# B&R Automation Studio project vibratorControlWithCurrentController (part 11)

#### producing.st
```iecst
ACTION producing:

	CASE em.state OF

		STATE_STARTING:

			em.cmd.sc := em.status.parent.state = STATE_STOPPING;

			CASE em.substate OF
				0:
					em.description := '';

					IF (NOT this.newRecipeLoaded AND interface.status.teachingDone AND this.brickCountTeached = recipe.brickCount) OR interface.cmd.skipTeach OR this.hmi.capconModeOff THEN
						interface.status.teachingDone := TRUE;
						brdkStrMemSet(ADR(this.pctFromMeanToLimit),0,SIZEOF(this.pctFromMeanToLimit));
						bufferIdxCounter :=0;
						this.MTDataStatistics_Teach(Enable:=FALSE);
						this.MTFilterMovingAverage_0(Enable:=FALSE);
						this.TeachIntegral_0.Enable := FALSE;
						this.TeachIntegral_0();
						em.substate := 100;
					ELSE
						interface.status.wingStartBrickNOK	:= TRUE;
						interface.parameter.teachBrickCount := 0;
						gCapconInterface.status.teachingDone := FALSE;
						gUpperFlapInterface.cmd.resetStatistics := TRUE; //
						gBottomFlapInterface.cmd.resetCassetteWaitTime := TRUE;
						brdkStrMemSet(ADR(this.pctFromMeanToLimit),0,SIZEOF(this.pctFromMeanToLimit));
						bufferIdxCounter :=0;
						this.countGoodPortionForTeach := 0;
						this.MTDataStatistics_1(Enable:=FALSE);
						this.MTDataStatistics_0(Enable:=FALSE);
						this.MTDataStatistics_Teach(Enable:=FALSE);
						this.MTFilterMovingAverage_0(Enable:=FALSE);
						this.TeachIntegral_0.Enable := FALSE;
						this.TeachIntegral_0();
						this.noAdaptiveTeaching := 0;
						interface.status.cycleTimeAutoMode := 0;
						gBeltInterface.cmd.cycleTimeCount := 0;
						this.MTFilterMovingAverage_1.Enable := FALSE;
						this.MTFilterMovingAverage_1();
						//always delete statistics before a new teach.
						resetStatistics;
						em.substate := 10;
					END_IF

				10:
					em.description := 'wait for wing to be ready';

					IF interface.cmd.wingReady OR interface.cmd.wingRequest THEN
						interface.status.ready := TRUE;
						em.substate := 20;
					END_IF

				20:
					em.description := 'wait for belt to feed bricks';

					IF gBeltInterface.status.dropBrickDone THEN
						interface.status.ready := FALSE;
						em.substate := 30;
					END_IF

				30:
					em.description := 'wait to see if brick is falling';

					this.TON_waitTime.IN := TRUE;
					this.TON_waitTime.PT := T#400ms;
					this.TON_waitTime();

					interface.status.wingStart := this.TON_waitTime.ET >= T#300ms;

					IF this.TON_waitTime.Q AND NOT interface.status.brickDetected THEN
						this.TON_waitTime.IN := FALSE;
						this.TON_waitTime();
						interface.status.wingStartBrickNOK := TRUE;
						em.substate := 40;
					END_IF

				40:
					em.description := 'wait for wing ready';

					IF interface.cmd.wingCmdAck OR gMainInterface.status.emptying THEN
						interface.status.wingStart := FALSE;
						interface.status.wingStartBrickNOK := FALSE;
						interface.status.wingStartBrickOK := FALSE;

						this.TeachIntegral_0.Enable 			:= TRUE;
						this.TeachIntegral_0.In 				:= interface.status.integralSum / USINT_TO_REAL(recipe.brickCount);
						this.TeachIntegral_0.BrickCount 		:= recipe.brickCount;
						this.TeachIntegral_0.CapconModeOn 		:= this.hmi.capconModeOn;
						this.TeachIntegral_0.NoPeaks 			:= interface.status.noVerifiedPeaks;
						this.TeachIntegral_0.NoPortions			:= config.portionsAllowTeach;
						this.TeachIntegral_0();

						interface.status.teachIntegral := this.TeachIntegral_0.Out;

						IF this.TeachIntegral_0.Done THEN
							this.TeachIntegral_0.Enable := FALSE;
							this.TeachIntegral_0();
							interface.status.teachingDone := TRUE;
							this.newRecipeLoaded := FALSE;
							em.substate := 100;
						ELSIF this.TeachIntegral_0.Error THEN
							this.TeachIntegral_0.Enable := FALSE;
							this.TeachIntegral_0();
							em.substate := 200;
						ELSE
							em.substate := 10;
						END_IF
					END_IF

				100:
					em.description := 'Wait for bypassCassette OFF';

					IF NOT gMainInterface.line.bypassCassette OR gMainInterface.status.emptying THEN
						em.substate := 110;
					END_IF

				110:
					em.description := 'teaching done';
					this.brickCountTeached := recipe.brickCount;
					em.cmd.sc := TRUE;

				200:
					em.description := 'teaching error';
					this.alarm.teachingError.active := TRUE;
					em.cmd.sc := TRUE;

			END_CASE

			// redo teaching if an empty is started while the reteach is running.
			IF interface.cmd.emptyWhileTeaching THEN
				this.hmi.redoTeaching := TRUE;
				em.cmd.sc := TRUE;
			END_IF

		STATE_EXECUTE:

			this.timeBetweenBricks := this.timeBetweenBricks + em.status.cycleTime;

			CASE em.substate OF
				0:
					em.description := 'wait for wing ready';

					interface.status.waiting := NOT interface.cmd.wingRequest;

					IF interface.cmd.wingRequest AND recipe.brickCount > 0 THEN
						IF recipe.brickCount <> this.brickCountTeached THEN
							this.newRecipeLoaded := TRUE;
						END_IF
						interface.status.ready := TRUE;
						em.cmd.sc := FALSE;
						this.startTime := 0;
						em.substate := 10;
					ELSE
						em.cmd.sc := TRUE;
					END_IF

				10:
					em.description := 'wait for belt to feed bricks';

					IF interface.cmd.wingReady AND this.startTime = 0 THEN
						this.startTime := TIME_TO_UDINT(clock_ms());
					END_IF

					IF gBeltInterface.status.dropBrickDone THEN
						interface.status.ready := FALSE;
						this.brickPresent := FALSE;
						IF this.startTime = 0 THEN
							this.startTime := TIME_TO_UDINT(clock_ms());
						END_IF
						em.substate := 20;
					END_IF

				20:
					em.description := 'wait to see if brick is falling';

					this.TON_waitTime.IN := TRUE;
					this.TON_waitTime.PT := T#400ms; // falltime through capcon is 400ms
					this.TON_waitTime();

					interface.status.wingStart := this.TON_waitTime.ET >= T#250ms;

					IF this.TON_waitTime.Q AND NOT interface.status.brickDetected THEN
						this.TON_waitTime.IN := FALSE;
						this.TON_waitTime();
						interface.status.wingStart := TRUE;

						em.substate := 30;
					END_IF

				30:
					em.description := 'validate brick';

					IF this.hmi.capconModeOff THEN
						// If capcon off = always OK capcon is completly OFF
						interface.status.wingStartBrickOK := TRUE;

						em.substate := 40;
//					ELSIF NOT gBeltInterface.status.gapOK AND (gBeltInterface.status.autoMode OR gBeltInterface.status.autoModeSimple) THEN
//						interface.status.wingStartBrickNOK := TRUE;
//						em.substate := 40;
					ELSIF interface.status.noVerifiedPeaks > interface.status.numBricksInPortion THEN
						this.hmi.count.integral.tooBig := this.hmi.count.integral.tooBig + 1;
						this.hmi.totalCount.integral.tooBig := this.hmi.totalCount.integral.tooBig + 1;
						interface.status.wingStartBrickNOK := TRUE;
						gBeltInterface.cmd.afterCount := NOT this.lastAfterCount;
						this.lastAfterCount := TRUE;
						em.substate := 40;
					ELSIF interface.status.noVerifiedPeaks < interface.status.numBricksInPortion AND this.hmi.capconModeOn THEN // only use lowerLimit if capconMode = ON
						this.hmi.count.integral.tooSmall := this.hmi.count.integral.tooSmall + 1;
						this.hmi.totalCount.integral.tooSmall := this.hmi.totalCount.integral.tooSmall + 1;
						interface.status.wingStartBrickNOK := TRUE;
						em.substate := 40;
					ELSE
						interface.status.wingStartBrickOK := TRUE;
						this.lastAfterCount := FALSE;
						em.substate := 40;
					END_IF

					this.totalTime := this.totalTime + (TIME_TO_UDINT(clock_ms())-this.startTime) + (MAX(MAX(gUpperFlapInterface.status.openCloseTime, gMiddleFlapInterface.status.openCloseTime), gBottomFlapInterface.status.openCloseTime)/1000);
					IF interface.status.wingStartBrickOK THEN

						this.MTFilterMovingAverage_0.Enable := TRUE;
						this.MTFilterMovingAverage_0.In := UDINT_TO_REAL(this.totalTime);
						this.MTFilterMovingAverage_0.WindowLength := 10;
						this.MTFilterMovingAverage_0();

						this.hmi.cycleTime := 60000/this.MTFilterMovingAverage_0.Out;
						this.hmi.cycleTimeTMU := this.MTFilterMovingAverage_0.Out/36;

						this.MTFilterMovingAverage_1.Enable := TRUE;
						this.MTFilterMovingAverage_1.In := UDINT_TO_REAL(this.totalTime);
						this.MTFilterMovingAverage_1.WindowLength := 20;
						this.MTFilterMovingAverage_1();

						interface.status.cycleTimeAutoMode := 60000/this.MTFilterMovingAverage_1.Out;
						gBeltInterface.cmd.cycleTimeCount := gBeltInterface.cmd.cycleTimeCount + 1;

						this.totalTime := 0;
					END_IF

					IF this.noAdaptiveTeaching < 8 OR this.newRecipeLoaded THEN

						this.TeachIntegral_0.Enable 			:= TRUE;
						this.TeachIntegral_0.In 				:= interface.status.integralSum / USINT_TO_REAL(recipe.brickCount);
						this.TeachIntegral_0.BrickCount 		:= recipe.brickCount;
						this.TeachIntegral_0.CapconModeOn 		:= this.hmi.capconModeOn;
						this.TeachIntegral_0.NoPeaks 			:= interface.status.noAdaptiveVerifiedPeaks;
						this.TeachIntegral_0.NoPortions			:= 3;
						this.TeachIntegral_0();

						interface.status.adaptiveTeachIntegral := this.TeachIntegral_0.Out;

						IF this.TeachIntegral_0.Done THEN
							this.TeachIntegral_0.Enable := FALSE;
							this.TeachIntegral_0();
							this.MTDataStatistics_0.In := this.TeachIntegral_0.Out;
							this.MTDataStatistics_0.Enable := TRUE;
							this.MTDataStatistics_0.MovingWindowLength := 8;
							this.MTDataStatistics_0();
							this.noAdaptiveTeaching := this.noAdaptiveTeaching + 1;
							IF this.newRecipeLoaded THEN
								this.newRecipeLoaded := FALSE;
								this.brickCountTeached := recipe.brickCount;
								this.countGoodPortionForTeach := 0;
								this.MTDataStatistics_1(Enable:=FALSE);
								interface.status.teachIntegral := this.TeachIntegral_0.Out;
								this.noAdaptiveTeaching := 0;
							ELSE
								interface.status.teachIntegral := this.MTDataStatistics_0.Mean;
							END_IF
						ELSIF this.TeachIntegral_0.Error THEN
							this.TeachIntegral_0.Enable := FALSE;
							this.TeachIntegral_0();
							IF this.newRecipeLoaded THEN
								this.alarm.teachingError.active := TRUE;
							END_IF
						END_IF

						IF interface.status.wingStartBrickOK THEN
							this.MTDataStatistics_Teach.In := interface.status.integralSum/USINT_TO_REAL(recipe.brickCount);
							this.MTDataStatistics_Teach.Enable := TRUE;
							this.MTDataStatistics_Teach.MovingWindowLength := 40;
							this.MTDataStatistics_Teach();
						END_IF

					ELSIF this.noAdaptiveTeaching >= 8 THEN

						IF interface.status.wingStartBrickOK THEN
							this.MTDataStatistics_Teach.In := interface.status.integralSum/USINT_TO_REAL(recipe.brickCount);
							this.MTDataStatistics_Teach.Enable := TRUE;
							this.MTDataStatistics_Teach.MovingWindowLength := 40;
							this.MTDataStatistics_Teach();

							this.hmi.capconMean := this.MTDataStatistics_Teach.Mean;
							this.hmi.capconMax := this.MTDataStatistics_Teach.MaxValue;
							this.hmi.capconMin := this.MTDataStatistics_Teach.MinValue;
							this.hmi.capconVariance := this.MTDataStatistics_Teach.Variance;
							this.hmi.integralSum := interface.status.integralSum;

							//
							IF this.countGoodPortionForTeach < 100 THEN
								this.MTDataStatistics_1.In := interface.status.integralSum/USINT_TO_REAL(recipe.brickCount);
								this.MTDataStatistics_1.Enable := TRUE;
								this.MTDataStatistics_1.MovingWindowLength := 40;
								this.MTDataStatistics_1();

								this.countGoodPortionForTeach := this.countGoodPortionForTeach + 1;
								IF this.countGoodPortionForTeach = 100 THEN
									// If 100 good portions - update teach integral to mean
									interface.status.teachIntegral := this.MTDataStatistics_1.Mean;
								END_IF
							END_IF
						END_IF

					END_IF

				40:
					em.description := 'wait for wing ready';

					IF interface.cmd.wingCmdAck OR gMainInterface.status.emptying THEN
						IF interface.status.wingStartBrickOK THEN
							this.hmi.count.portions.count := this.hmi.count.portions.count + 1;
							this.hmi.totalCount.portions.count := this.hmi.totalCount.portions.count + 1;
						ELSIF interface.status.wingStartBrickNOK THEN
							this.hmi.count.reject.count := this.hmi.count.reject.count + 1;
							this.hmi.totalCount.reject.count := this.hmi.totalCount.reject.count + 1;
						END_IF
						this.hmi.count.total := this.hmi.count.portions.count + this.hmi.count.reject.count;
						this.hmi.totalCount.total := this.hmi.totalCount.portions.count + this.hmi.totalCount.reject.count;
						IF this.hmi.count.total > 0 THEN
							tmpCal := UDINT_TO_REAL(this.hmi.count.portions.count) / UDINT_TO_REAL(this.hmi.count.total);
							this.hmi.count.portions.percent := tmpCal * 100.0;
							this.hmi.count.reject.percent := 100.0-this.hmi.count.portions.percent;
						END_IF
						this.lastPortionOK := interface.status.wingStartBrickOK;
						interface.status.wingStart 			:= FALSE;
						interface.status.wingStartBrickNOK 	:= FALSE;
						interface.status.wingStartBrickOK 	:= FALSE;
						gBeltInterface.cmd.afterCount := FALSE;
						em.substate := 0;
					END_IF

			END_CASE

			em.cmd.sc := TRUE;

		STATE_COMPLETING:

			interface.status.ready := interface.cmd.wingRequest;

			CASE em.substate OF
				0:
					em.description := 'Waiting for wing to be ready';
					IF interface.cmd.wingRequest THEN
						interface.status.wingStartBrickNOK	:= TRUE;
						em.substate := 10;
					END_IF

				10:
					em.description := 'Waiting wing to ack reject command';

					IF interface.cmd.wingCmdAck THEN
						interface.status.wingStartBrickNOK	:= FALSE;
						em.substate := 0;
					END_IF
			END_CASE

			em.cmd.sc := interface.cmd.emptyStop;

		STATE_SUSPENDED:

			em.description := 'wing ready to receive drop';
			interface.status.ready := interface.cmd.wingReady AND NOT interface.cmd.brickIncomming;
			interface.status.waiting := NOT interface.cmd.wingReady;
			em.cmd.sc := TRUE;

		STATE_ABORTED:

			IF NOT MpAlarmXCheckReaction(mpAlarmXCore,'abortCapcon') THEN
				em.cmd.sc := TRUE;
			END_IF

		STATE_CLEARING:

			brsmemset(ADR(this.alarm), 0, SIZEOF(this.alarm));
			//Alarm texts
			this.alarm.teachingError.name := 'capconTeachingError';

			em.cmd.sc := TRUE;

		STATE_STOPPED:

			em.description := 'Waiting for start command';

			IF gConfig.status.loadInitialValue[3] AND (gRecipe.status.saved OR gRecipe.status.loaded) AND (gConfig.status.saved OR gConfig.status.loaded) THEN
				gConfig.status.loadInitialValue[3] := FALSE;
				recipe.brickCount := 1;
				recipe.controlPrc := 45;
			END_IF
			em.cmd.sc := TRUE;

		STATE_STOPPING, STATE_ABORTING:
			interface.status.ready := FALSE;
			this.hmi.cycleTime := 0;
			this.hmi.cycleTimeTMU := 0;
			interface.status.cycleTimeAutoMode := 0;
			gBeltInterface.cmd.cycleTimeCount := 0;
			interface.status.wingStartBrickNOK := FALSE;
			interface.status.wingStartBrickOK := FALSE;
			interface.status.wingStart := FALSE;
			em.cmd.sc := TRUE;

		ELSE

			em.cmd.sc := TRUE;

	END_CASE

END_ACTION
```

#### alarm.st
```iecst
ACTION alarm:

	// Teaching Error

	IF this.alarm.teachingError.active AND NOT this.alarm.teachingError.oldActive THEN
		this.alarm.teachingError.instanceID := MpAlarmXSet(mpAlarmXCore, this.alarm.teachingError.name);
	END_IF
	this.alarm.teachingError.oldActive := this.alarm.teachingError.active;

	// Alarms are also set in sampling task

	(****************************** REACTION ******************************)
	IF em.state <> STATE_ABORTED AND em.state <> STATE_ABORTING AND em.state <> STATE_CLEARING THEN
		IF MpAlarmXCheckReaction(mpAlarmXCore,'abortCapcon') THEN
			em.cmd.abort := TRUE;
		END_IF
	END_IF
	(**********************************************************************)

END_ACTION
```

#### capcon.st - Init, cyclic, exit code
```iecst
PROGRAM _INIT

	em.setup.name := 'capcon';
	em.setup.parent.name := 'main';
	em.setup.lastActivated := FALSE;

	// gets the task name and setup names for config and receipe types
	ST_name(0,ADR(this.names.configName),0);
	brdkStrCpy(ADR(this.names.recipeName),ADR(this.names.configName));
	brdkStrCpy(ADR(this.names.recipeNameCurrent),ADR(this.names.configName));
	brdkStrCat(ADR(this.names.configName),ADR(':this.hmi.config'));
	brdkStrCat(ADR(this.names.recipeName),ADR(':this.hmi.recipe'));
	brdkStrCat(ADR(this.names.recipeNameCurrent),ADR(':this.hmi.recipeCurrent'));

	setupPointers;

	//Alarm texts
	this.alarm.teachingError.name := 'capconTeachingError';

END_PROGRAM

PROGRAM _CYCLIC

	setupPointers;

	IF gRecipe.status.newRecipeLoaded OR this.hmi.redoTeaching OR interface.cmd.reTeach THEN
		interface.cmd.reTeach := FALSE;
		gRecipe.status.newRecipeLoaded 	:= FALSE;
		this.hmi.redoTeaching			:= FALSE;
		this.newRecipeLoaded 			:= TRUE;
	END_IF

	interface.parameter.simSampleDelay 	:= config.simSampleDelay;
	interface.parameter.controlPercent 	:= recipe.controlPrc;
	interface.parameter.capconMode 		:= recipe.capconMode;
	interface.status.cycleTime 			:= em.status.cycleTime;
	brsmemcpy(ADR(interface.config),ADR(config),SIZEOF(interface.config));

	countersData := countersData;
	TMU := TMU;

	CASE em.mode OF
		MODE_PRODUCING: producing;
		ELSE em.cmd.sc := TRUE;
	END_CASE

	alarm;

	em();

	interface.status.wingDosing := gRecipe.status.loaded AND (recipe.brickCount = 0 OR gMainInterface.line.bypassCassette);
	interface.status.numBricksInPortion := USINT_TO_UDINT(recipe.brickCount);
	interface.status.factorRmsMax := config.factorRmsMax;
	interface.status.capconMinThreshold := config.capconMinThreshold;

	// copy the recipe data
	CASE interface.cmd.copyRecipe OF

		COPY_RECIPE_NEXT_TO_WORKING:
			IF gMainInterface.cmd.loadingTemplateRecipe THEN
				gMainInterface.cmd.loadingTemplateRecipe := FALSE;
				// Template recipe can't load brickCount
				this.brickCount := this.hmi.recipe.brickCount;
				this.hmi.recipe := this.hmi.recipeCurrent;
				this.hmi.recipe.brickCount := this.brickCount;
			ELSE
				this.hmi.recipe := this.hmi.recipeCurrent;
			END_IF

			//	this.hmi.recipe.controlPrcIdx := LIMIT(0, REAL_TO_USINT((USINT_TO_REAL(this.hmi.recipe.controlPrc)-35.0) / 10.0), 5);

			recipe.controlPrc := 45;
			recipe.controlPrcIdx := 1;
			recipe.controlPrcOld := 45;
			interface.status.numBricksInPortion := USINT_TO_UDINT(recipe.brickCount);
			gBeltInterface.cmd.initRecipe := TRUE; // Belt can only init when we know brickcount.
			gVibratorInterface[0].cmd.initRecipe := gVibratorInterface[1].cmd.initRecipe := TRUE; // Vibrator can only init recipe when we know brickcount
			gRecipe.cmd.save 			:= TRUE;
			interface.cmd.copyRecipe 	:= COPY_RECIPE_NONE;

		COPY_RECIPE_SANDBOX_TO_NEXT:
			interface.cmd.copyRecipe 	:= COPY_RECIPE_NONE;

	END_CASE

	// Convert control% dropdown to controlPrc
	CASE this.hmi.recipe.controlPrcIdx OF
		0:
			this.hmi.recipe.controlPrc := 35;
		1:
			this.hmi.recipe.controlPrc := 45;
		2:
			this.hmi.recipe.controlPrc := 55;
		3:
			this.hmi.recipe.controlPrc := 65;
		4:
			this.hmi.recipe.controlPrc := 75;
		5:
			this.hmi.recipe.controlPrc := 85;
		ELSE
			this.hmi.recipe.controlPrc := 0;
	END_CASE

	IF gRecipe.status.doCheckForChanges AND NOT this.oldCheckChangesRecipe THEN
		gMainInterface.status.statusIT.PortionItemCount := USINT_TO_INT(recipe.brickCount);
		this.MpRecipeRegPar_Recipe.Enable := TRUE;
		this.MpRecipeRegPar_RecipeCurrent.Enable := TRUE;

		IF gRecipe.status.loaded AND NOT this.oldLoadedRecipe THEN
			// Initial program load. Set old=new to avoid saving just after a load (makes no sense)
			this.recipeOld := this.hmi.recipe;
		END_IF
		this.oldLoadedRecipe := gRecipe.status.loaded;

		IF NOT gRecipe.cmd.save AND gRecipe.status.loaded AND (brsmemcmp(ADR(this.hmi.recipe),ADR(this.recipeOld),SIZEOF(this.recipeOld)) <> 0) THEN
			gRecipe.cmd.save := TRUE;
			this.recipeOld := this.hmi.recipe;
		END_IF

	END_IF
	this.MpRecipeRegPar_Recipe(MpLink := ADR(mpRecipe), PVName := ADR(this.names.recipeName), Category := ADR('recipe'));
	this.MpRecipeRegPar_RecipeCurrent(MpLink := ADR(mpRecipeCurrent), PVName := ADR(this.names.recipeNameCurrent), Category := ADR('recipeCurrent'));
	this.oldCheckChangesRecipe := gRecipe.status.doCheckForChanges;

	IF gConfig.status.doCheckForChanges AND NOT this.oldCheckChangesConfig THEN
		this.MpRecipeRegPar_Config.Enable := TRUE;

		IF gConfig.status.loaded AND NOT this.oldLoaded THEN
			// Initial program load. Set old=new to avoid saving just after a load (makes no sense)
			this.configOld := this.hmi.config;
		END_IF
		this.oldLoaded := gConfig.status.loaded;

		IF NOT gConfig.cmd.save AND gConfig.status.loaded AND (brsmemcmp(ADR(this.hmi.config),ADR(this.configOld),SIZEOF(this.configOld)) <> 0) THEN
			gConfig.cmd.save := TRUE;
			this.configOld := this.hmi.config;
		END_IF

	END_IF
	this.MpRecipeRegPar_Config(MpLink := ADR(mpRecipe), PVName := ADR(this.names.configName), Category := ADR('config'));
	this.oldCheckChangesConfig := gConfig.status.doCheckForChanges;

	// Calculate count percentages
	this.sumStatistik := UDINT_TO_REAL(this.hmi.count.integral.tooBig + this.hmi.count.integral.tooSmall + this.hmi.count.invalidBuffer.count + gUpperFlapInterface.status.countAftercount);

	this.hmi.capconModeOn 		:= this.hmi.recipe.capconMode = 0;
	this.hmi.capconModeMedium 	:= this.hmi.recipe.capconMode = 1;
	this.hmi.capconModeOff 		:= this.hmi.recipe.capconMode = 2;
	this.hmi.teaching			:= this.newRecipeLoaded AND (em.state = STATE_STARTING OR em.state = STATE_EXECUTE);

	IF this.sumStatistik = 0 THEN
		this.hmi.count.integral.tooBigPercent	:= 0;
		this.hmi.count.integral.tooSmallPercent	:= 0;
		this.hmi.count.afterCounting.percent	:= 0;
		this.hmi.count.invalidBuffer.percent	:= 0;
		gUpperFlapInterface.status.countAftercount := 0; // only upperFlap knows the amount of aftercounts.
	ELSE
		this.hmi.count.integral.tooBigPercent	:= UDINT_TO_REAL(this.hmi.count.integral.tooBig) / this.sumStatistik * 100;
		this.hmi.count.integral.tooSmallPercent	:= UDINT_TO_REAL(this.hmi.count.integral.tooSmall) / this.sumStatistik * 100;
		this.hmi.count.afterCounting.percent	:= UDINT_TO_REAL(gUpperFlapInterface.status.countAftercount) / this.sumStatistik * 100;
		this.hmi.count.invalidBuffer.percent	:= UDINT_TO_REAL(this.hmi.count.invalidBuffer.count) / this.sumStatistik * 100;
	END_IF;

	interface.status.state := em.state;

	IF gConfig.status.factoryReset[3] THEN
		gConfig.status.factoryReset[3] := FALSE;
		// Factory reset all parameters:
		config.noStopDelay := 100;
		config.logToFile := FALSE;
		config.capconNoiseAllowedPeakToPeak := 55;
		config.capconDcOffsetAllowed := 800;
		config.capconNoiseAllowedSpeed := 2000;
		config.simSampleDelay := 150;
		config.portionsAllowTeach := 10;

		recipe.controlPrc := 55;
		recipe.controlPrcOld := 55;
		recipe.capconMode := 0;
		recipe.controlPrcIdx := 2;
	END_IF
END_PROGRAM

PROGRAM _EXIT
	setupPointers;
	this.MpRecipeRegPar_Recipe(Enable := FALSE);
	this.MpRecipeRegPar_Config(Enable := FALSE);
	this.MpRecipeRegPar_RecipeCurrent(Enable := FALSE);
END_PROGRAM
```

#### setupPointers.st
```iecst
ACTION setupPointers:
	recipe ACCESS ADR(this.hmi.recipe);
	config ACCESS ADR(this.hmi.config);
	interface ACCESS ADR(gCapconInterface);
END_ACTION
```

#### local.typ - Local data types
```iecst
TYPE
	counters_data_typ : 	STRUCT
		itemAfterCounting : UDINT;
		itemCountToFew : UDINT;
		itemCountToMany : UDINT;
		itemSizeToLarge : UDINT;
		itemSizeToSmall : UDINT;
		okCount : UDINT;
	END_STRUCT;
	local_updateHMIandRecord : 	STRUCT
		MpDataRegPar : ARRAY[0..19]OF MpDataRegPar;
		state : USINT;
		updateCmd : BOOL;
		length : DINT;
		lengthNew : DINT;
		startIdx : DINT;
		record : local_record_typ;
	END_STRUCT;
	recipe_capcon_typ : 	STRUCT
		controlPrcOld : USINT := 55; (*%*)
		brickCount : USINT := 1;
		controlPrc : USINT := 55;
		controlPrcIdx : USINT := 2;
		capconMode : USINT := 0; (*0: On, 1: Medium, 2: Off*)
	END_STRUCT;
	local_typ : 	STRUCT
		hmi : hmi_typ;
		alarm : local_alarm_typ;
		MpRecipeRegPar_Config : MpRecipeRegPar;
		MpRecipeRegPar_Recipe : MpRecipeRegPar;
		MpRecipeRegPar_RecipeCurrent : MpRecipeRegPar;
		time : local_time_typ;
		integral : REAL;
		samples : UDINT;
		topAvgSignal : REAL;
		emptyRejectCount : USINT;
		TON_timeout : TON;
		configOld : config_capcon_typ;
		recipeOld : recipe_capcon_typ;
		useTeachCount : UDINT;
		sumStatistik : REAL;
		timeBetweenBricks : UDINT;
		newRecipeLoaded : BOOL;
		dropTimeIdx : USINT;
		droptimes : ARRAY[0..100]OF REAL;
		wingOldReady : BOOL;
		controlOld : USINT;
		names : local_names_typ;
		inCommingCount : INT;
		peakCount : USINT;
		moreThan2Peaks : BOOL; (*Capcon signal have more than 2 peaks. ONLY topMax strategy is valid if signal have > 1 peak*)
		rejectInPortion : BOOL; (*True if at least 1 reject in the portion. Will be reset after each portion.*)
		brickCount : USINT;
		TON_waitTime : TON;
		brickPresent : BOOL;
		lastPortionOK : BOOL;
		brickCountTeached : USINT; (*Brick count that we teached with.*)
		timeBrickIsFalling : TIME := T#400ms;
		pctFromMeanToLimit : ARRAY[0..MAX_PCT_FROM_MEAN]OF REAL;
		MTDataStatistics_Teach : MTDataStatistics;
		MTDataStatistics_0 : MTDataStatistics;
		MTDataStatistics_1 : MTDataStatistics;
		countGoodPortionForTeach : USINT;
		errorTeachCounter : USINT;
		newTeachMean : REAL;
		TeachIntegral_0 : TeachIntegral;
		startTime : UDINT;
		totalTime : UDINT;
		MTFilterMovingAverage_0 : MTFilterMovingAverage;
		noAdaptiveTeaching : UDINT;
		lastAfterCount : BOOL;
		oldCheckChangesConfig : BOOL;
		oldCheckChangesRecipe : BOOL;
		oldLoaded : BOOL;
		oldLoadedRecipe : BOOL;
		MTFilterMovingAverage_1 : MTFilterMovingAverage;
	END_STRUCT;
	hmi_typ : 	STRUCT
		config : config_capcon_typ;
		recipe : recipe_capcon_typ;
		actualBrickInPortion : UDINT;
		count : local_hmi_count_typ;
		totalCount : local_hmi_count_typ;
		previusError : STRING[80];
		lastError : STRING[80];
		pcsPerMin : REAL;
		tmu : REAL;
		ultilityPercent : REAL;
		integral : REAL;
		samples : UDINT;
		topAvgSignal : REAL;
		redoTeaching : BOOL;
		maxSpeedNoise : REAL;
		recipeCurrent : recipe_capcon_typ;
		capconModeMedium : BOOL;
		capconModeOff : BOOL;
		capconModeOn : BOOL;
		cycleTimeTMU : REAL;
		cycleTime : REAL;
		teaching : BOOL;
		capconMax : REAL;
		capconMin : REAL;
		capconMean : REAL;
		capconVariance : REAL;
		integralSum : REAL;
	END_STRUCT;
	local_time_typ : 	STRUCT
		elapsed : UDINT;
		maximum : UDINT;
	END_STRUCT;
	local_names_typ : 	STRUCT
		configName : STRING[80];
		recipeName : STRING[80];
		recipeNameCurrent : STRING[80];
	END_STRUCT;
	local_record_typ : 	STRUCT
		avgSignalData : ARRAY[0..CAPCON_LOG_SAMPLE_SIZE]OF REAL;
		avgSpeedData : ARRAY[0..CAPCON_LOG_SAMPLE_SIZE]OF REAL;
		rawData : ARRAY[0..CAPCON_LOG_SAMPLE_SIZE]OF INT;
		avgSignalPoints : ARRAY[0..2]OF REAL;
		avgSpeedPoints : ARRAY[0..2]OF REAL;
		idxPoints : ARRAY[0..2]OF DINT;
		integral : REAL;
		samples : UDINT;
		topAvgSignal : REAL;
		validation : local_element_validation_typ;
		count : UDINT;
	END_STRUCT;
	local_peak_typ : 	STRUCT
		currentNettime : DINT;
		start : local_peak_point_typ;
		top : local_peak_point_typ;
		end : local_peak_point_typ;
		count : REAL;
		buffers : local_peak_buffer_typ;
		internalCount : USINT;
		internalRejectCount : USINT;
	END_STRUCT;
	local_peak_point_typ : 	STRUCT
		nettime : DINT;
		value : REAL;
	END_STRUCT;
	local_peak_buffer_typ : 	STRUCT
		live : ARRAY[0..99]OF REAL; (*tmp live data buffer to be copied to peak buffer*)
		peak : ARRAY[0..99]OF REAL; (*buffer containing the last detected peak, time starts from 0 and ends with peakTimespan [ms]*)
		peakCountdownCpy : DINT; (*samples to wait before copying live to get a top more er less in the middle*)
		peakTimespan : UDINT; (*Timespan of the peak buffer in ms*)
		peakCursor2 : UDINT; (*Time of cursor 2 (peak end point) in ms from peak buffer start*)
		peakCursor1 : UDINT; (*Time of cursor 1 (peak end point) in ms from peak buffer start*)
	END_STRUCT;
	local_element_validation_typ :
		(
		CAPCON_VALIDATION_NONE := 0,
		CAPCON_VALIDATION_ACCEPT := 1,
		CAPCON_VAL_REJECT_SAMP_TOO_SMALL := 2,
		CAPCON_VAL_REJECT_SAMP_TOO_BIG := 3,
		CAPCON_VAL_REJECT_PEAK_TOO_SMALL := 4,
		CAPCON_VAL_REJECT_PEAK_TOO_BIG := 5,
		CAPCON_VAL_REJECT_INT_TOO_SMALL := 6,
		CAPCON_VAL_REJECT_INT_TOO_BIG := 7,
		CAPCON_VAL_REJECT_INVALID := 8,
		CAPCON_VAL_REJECT_AFTER_COUNT := 9,
		CAPCON_VAL_REJECT_TIMEOUT := 10,
		CAPCON_VAL_REJECT_TOO_MANY := 11
		) := CAPCON_VALIDATION_NONE;
	local_hmi_count_item_typ : 	STRUCT
		percent : REAL;
		count : UDINT;
	END_STRUCT;
	local_hmi_count_min_max_item_typ : 	STRUCT
		tooSmallPercent : REAL;
		tooBigPercent : REAL;
		tooSmall : UDINT;
		tooBig : UDINT;
	END_STRUCT;
	local_hmi_count_typ : 	STRUCT
		reject : local_hmi_count_item_typ;
		portions : local_hmi_count_item_typ;
		integral : local_hmi_count_min_max_item_typ;
		afterCounting : local_hmi_count_item_typ;
		invalidBuffer : local_hmi_count_item_typ;
		total : UDINT;
	END_STRUCT;
	config_capcon_typ : 	STRUCT
		noStopDelay : UDINT := 100; (*[ms] delay between two bricks that there is time to turn the reject system*)
		simSampleDelay : UDINT := 150; (*[ms] delay to when the sampleing is starting*)
		capconNoiseAllowedPeakToPeak : REAL := 55; (*[mV] noise we allow on passive capcon signal before throwing alarm.*)
		capconDcOffsetAllowed : REAL := 800; (*[mV] tolerance for DC-offset on signal before making an alarm*)
		logToFile : BOOL := FALSE;
		capconNoiseAllowedSpeed : REAL := 2000;
		factorRmsMax : REAL := 0.001;
		capconMinThreshold : REAL := 100.0;
		portionsAllowTeach : USINT := 10;
	END_STRUCT;
	local_alarm_typ : 	STRUCT
		teachingError : gAlarm_struct_typ;
	END_STRUCT;
	BUFFER_BRICK_STATE :
		(
		BUFFER_BRICK_END,
		BUFFER_BRICK_MIDDLE,
		BUFFER_BRICK_START
		);
END_TYPE
```

#### local.var - Local variables
```iecst
VAR CONSTANT
	MAX_TEACH_CANDIDATES : USINT := 15;
END_VAR
VAR
	countersData : counters_data_typ;
	interface : REFERENCE TO gCapconInterface_typ;
	tmpCal : REAL;
	i : DINT;
	this : {REDUND_UNREPLICABLE} local_typ;
	em : {REDUND_UNREPLICABLE} brdkEM;
	recipe : REFERENCE TO recipe_capcon_typ;
	config : REFERENCE TO config_capcon_typ;
END_VAR
VAR CONSTANT
	CAPCON_START_RECORD_SAMPLE_COUNT : DINT := 150; (*number of samples that is needed for a record before the start index *)
END_VAR
VAR
	TMU : UDINT;
END_VAR
VAR CONSTANT
	MAX_PCT_FROM_MEAN : USINT := 99;
END_VAR
VAR
	bufferIdxCounter : USINT;
END_VAR
```

#### LocalFunctions.fun
```iecst
{REDUND_ERROR} FUNCTION_BLOCK TeachIntegral (*TODO: Add your comment here*) (*$GROUP=User,$CAT=User,$GROUPICON=User.png,$CATICON=User.png*)
	VAR_INPUT
		Enable : {REDUND_UNREPLICABLE} BOOL;
		BrickCount : USINT;
		NoPeaks : USINT;
		CapconModeOn : BOOL;
		NoPortions : USINT; (*The amount of good portions that have to be seen before accepting teach*)
		In : REAL;
	END_VAR
	VAR_OUTPUT
		Out : REAL;
		Done : BOOL;
		Error : BOOL;
	END_VAR
	VAR
		teachCandidate : {REDUND_UNREPLICABLE} BOOL;
		teachCandidateIntegral : ARRAY[0..MAX_TEACH_CANDIDATES] OF REAL;
		teachIntegral : REAL;
		teachCandidateCounter : USINT;
		teachCounter : USINT;
		state : UINT;
		i : UINT;
	END_VAR
END_FUNCTION_BLOCK
```

#### LocalFunctions.st
```iecst
FUNCTION_BLOCK TeachIntegral

	CASE state OF
		0:
			IF Enable THEN
				IF NOT teachCandidate THEN
					teachCandidateIntegral[0] := In;
					Out := In;
					teachCandidateCounter := 1;
					teachCandidate := TRUE;
				ELSE
					IF NoPeaks <> BrickCount AND CapconModeOn THEN
						teachCandidate := FALSE;
						teachCandidateCounter := 0;
						teachCounter := teachCounter + 1;
						IF teachCounter = 18 THEN
							state := 100;
						END_IF
					ELSE
						teachCandidateIntegral[teachCandidateCounter] := In;
						teachCandidateCounter := teachCandidateCounter + 1;
						IF teachCandidateCounter > MIN(MAX_TEACH_CANDIDATES, NoPortions) THEN
							teachIntegral := 0;
							FOR i:=0 TO MAX_TEACH_CANDIDATES DO
								teachIntegral := teachIntegral + teachCandidateIntegral[i];
							END_FOR
							teachIntegral := teachIntegral / USINT_TO_REAL(MIN(MAX_TEACH_CANDIDATES, NoPortions)+1);
							state := 10;
						END_IF
					END_IF
				END_IF
			END_IF

		10:
			Done := TRUE;

		100:
			Error := TRUE;

	END_CASE

	IF NOT Enable THEN
		Done := FALSE;
		Error := FALSE;
		brsmemset(ADR(teachCandidateIntegral), 0, SIZEOF(teachCandidateIntegral));
		teachCandidate := FALSE;
		teachIntegral := 0;
		state := 0;
	END_IF

END_FUNCTION_BLOCK
```

#### resetStatistics.st
```iecst
ACTION resetStatistics:
	this.hmi.count.integral.tooBig := 0;
	this.hmi.count.integral.tooSmall := 0;
	//this.hmi.count.peak.tooBig := 0;
	//this.hmi.count.peak.tooSmall := 0;
//	this.hmi.count.samples.tooBig := 0;
//	this.hmi.count.samples.tooSmall := 0;
	gUpperFlapInterface.status.countAftercount := 0;
	this.hmi.count.invalidBuffer.count := 0;
	this.hmi.count.portions.count := 0;
//	this.hmi.count.timeouts.count := 0;
	this.hmi.count.reject.percent := 0;
	this.hmi.count.reject.count := 0;
END_ACTION
```

### capconGlobal.typ
```iecst
TYPE
	gCapconInterface_typ : 	STRUCT
		cmd : gCapconInterface_cmd_typ;
		status : gCapconInterface_status_typ;
		parameter : gCapconInterface_par_typ;
		config : gCapconInterface_config_typ;
	END_STRUCT;
	gCapconInterface_config_typ : 	STRUCT
		speedMinLimit : REAL; (*indicates the speed min limit for when you are sure that a brick has passed through*)
		speedMaxLimit : REAL; (*indicates the speed max limit for when you are sure that a brick has passed through*)
		noStopDelay : UDINT; (*[ms] delay between two bricks that there is time to turn the reject system*)
		simSampleDelay : UDINT := 150; (*[ms] delay to when the sampleing is starting*)
		brickIncomingTimeout : UDINT := 1000; (*[ms] timeout signal from when a brick was incomming*)
		capconNoiseAllowedPeakToPeak : REAL := 55; (*[mV] noise we allow on passive capcon signal before throwing alarm.*)
		capconDcOffsetAllowed : REAL := 800; (*[mV] tolerance for DC-offset on signal before making an alarm*)
		logToFile : BOOL;
		capconNoiseAllowedSpeed : REAL;
	END_STRUCT;
	gCapconInterface_cmd_typ : 	STRUCT
		resetCounters : BOOL;
		startLogging : BOOL;
		portionIncomming : BOOL;
		brickIncomming : BOOL;
		calculateStatistics : BOOL;
		skipTeach : BOOL;
		emptyStop : BOOL;
		wingReady : BOOL;
		wingRequest : BOOL;
		wingCmdAck : BOOL;
		startTeaching : BOOL;
		emptyWhileTeaching : BOOL;
		copyRecipe : copy_recipe_command_typ;
		reTeach : BOOL;
		startSpeedSignalTest : BOOL;
	END_STRUCT;
	teach_status_typ : 	STRUCT
		maxSpeed : ARRAY[0..CAPCON_TEACH_BRICK_COUNT]OF REAL;
		integral : ARRAY[0..CAPCON_TEACH_BRICK_COUNT]OF REAL;
		topAvgSignal : ARRAY[0..CAPCON_TEACH_BRICK_COUNT]OF REAL;
		samples : ARRAY[0..CAPCON_TEACH_BRICK_COUNT]OF UDINT;
		brickDetected : BOOL;
	END_STRUCT;
	gCapconInterface_par_limit_typ : 	STRUCT
		maxSamples : UDINT;
		minSamples : UDINT;
		maxTop : REAL;
		minTop : REAL;
		maxIntegral : REAL;
		minIntegral : REAL;
	END_STRUCT;
	gCapconInterface_par_typ : 	STRUCT
		limits : gCapconInterface_par_limit_typ;
		teachBrickCount : UDINT := 0;
		count : UDINT;
		controlPercent : USINT;
		simSampleDelay : UDINT;
		brickCount : USINT;
		capconMode : USINT;
	END_STRUCT;
	gCapconInterface_status_typ : 	STRUCT
		ready : BOOL;
		teach : teach_status_typ;
		teachingDone : BOOL;
		waiting : BOOL;
		cycleTime : UDINT;
		reset : BOOL;
		wingStartBrickNOK : BOOL;
		wingStartBrickOK : BOOL;
		state : brdk_em_states_typ;
		wingDosing : BOOL;
		numBricksInPortion : UDINT;
		maxNoiseSpeed : REAL;
		integralSum : REAL;
		brickDetected : BOOL;
		brickPresent : BOOL;
		noPeaks : USINT;
		noVerifiedPeaks : USINT;
		teachIntegral : REAL;
		adaptiveTeachIntegral : REAL;
		noAdaptiveVerifiedPeaks : USINT;
		wingStart : BOOL;
		verifiedPeakCount : ARRAY[0..MAX_PEAKS]OF USINT;
		peakIntegral : ARRAY[0..MAX_PEAKS]OF REAL;
		factorRmsMax : REAL;
		capconMinThreshold : REAL;
		cycleTimeAutoMode : REAL;
		maxRawSignal : REAL;
	END_STRUCT;
	gCapconBufferResult_typ : 	STRUCT
		samples : UDINT;
		integral : REAL;
		topAvgSignal : REAL;
		done : BOOL;
		peakValue : ARRAY[0..CAPCON_MAX_PEAK_COUNT]OF REAL;
		maxSpeed : REAL;
		peakCount : USINT;
	END_STRUCT;
	gCapcon_buffer_typ : 	STRUCT
		sample : ARRAY[0..CAPCON_MAX_BUFFER_SIZE]OF gCapcon_buffer_sample_typ;
		idx : DINT;
		topIdx : ARRAY[0..CAPCON_MAX_PEAK_COUNT]OF DINT;
		startIdx : DINT;
		endIdx : DINT;
		active : BOOL;
		invalid : BOOL;
		startTopSampleRange : DINT;
		endTopSampleRange : DINT;
		new : BOOL;
		notAbrick : BOOL;
		nextBrick : BOOL;
		result : gCapconBufferResult_typ;
		nextBrickStart : INT;
	END_STRUCT;
	gCapcon_buffer_sample_typ : 	STRUCT
		avgSpeed : REAL;
		avgSignal : REAL;
		raw : INT;
	END_STRUCT;
END_TYPE
```

### capconGlobal.var
```iecst
VAR CONSTANT
	MAX_PEAKS : USINT := 29;
END_VAR
VAR
	gCapconInterface : gCapconInterface_typ;
END_VAR
VAR CONSTANT
	CAPCON_TEACH_BRICK_COUNT : UINT := 99; (*The amount of bricks to measure during teaching. 9 means 10*)
	CAPCON_MAX_BUFFER_SIZE : DINT := 999; (*Max size of capcon buffer. 999 means 1000*)
	CAPCON_MAX_PEAK_COUNT : USINT := 9; (*9 means 10. Max. number of peaks in a signal*)
END_VAR
```

### Program Logical/modules/main/wing/wing (IEC)

#### producing.st
```iecst
ACTION producing:

	CASE em.state OF

		STATE_STOPPED:
			em.description 			:= 'start wing unit right away';

			IF gUpperFlapInterface.status.active AND gMiddleFlapInterface.status.active AND gBottomFlapInterface.status.active THEN
				// start wing as soon as all childs are active (they are active when they enter STATE_STOPPED).
				this.time.elapsed := this.time.elapsed + em.status.cycleTime;
				IF this.time.elapsed >= 2000000 THEN
					// Wait 2s before we start.
					em.cmd.sc 				:= TRUE;
					em.cmd.reset			:= TRUE;
				END_IF
			ELSE
				this.time.elapsed := 0;
			END_IF

		STATE_IDLE:
			em.description 	:= 'wing unit must always be started';
			em.cmd.sc := em.cmd.start 		:= TRUE;

		STATE_STARTING:
			em.description := 'waiting for ready command from upper flap';
//
				interface.status.ready 	:= TRUE;
				interface.cmd.startManuelMode := FALSE;

				this.cycleTime		:= 0;
				this.cycleTimeIdx	:= 0;
				this.waitingTimeIdx	:= 0;
				this.hmi.cycleTime := 0;
				this.hmi.cycleTimeTmu := 0;
				this.hmi.waitTimeUtilisation := 0;
				brdkStrMemSet(ADR(this.cycleTimes),0,SIZEOF(this.cycleTimes));
				brdkStrMemSet(ADR(this.cycleTimesTmu),0,SIZEOF(this.cycleTimesTmu));
				brdkStrMemSet(ADR(this.waitingTimeBuffer),0,SIZEOF(this.waitingTimeBuffer));

				interface.status.request := TRUE;
				this.utilityBufferActive := FALSE;

				IF gCapconInterface.status.teachingDone THEN
					this.blockCycleTime := TRUE;
				ELSE
					this.blockCycleTime := FALSE;
				END_IF

				this.oldEmptyMode := interface.cmd.shaftModeEmpty; // To avoid delay on first start. Only relevant when changing mode doing STATE_EXECUTE.
				em.cmd.sc 	:= TRUE;

		STATE_EXECUTE:

			interface.status.ready := gUpperFlapInterface.status.ready;

			em.description 									:= 'waiting for commands';

			IF interface.cmd.startBrick AND NOT interface.status.commandAck THEN
				gUpperFlapInterface.cmd.start 				:= TRUE;
				interface.status.ready 						:= FALSE;
				interface.status.request					:= FALSE;
				interface.status.commandAck					:= TRUE;
			END_IF

			IF (interface.cmd.startBrickOK OR interface.cmd.startBrickNOK) AND NOT gUpperFlapInterface.cmd.brickStatusReady THEN
				gUpperFlapInterface.parameter.brickStatus 	:= SEL(interface.cmd.startBrickNOK, BRICK_STATUS_OK, BRICK_STATUS_NOK);
				gUpperFlapInterface.cmd.brickStatusReady 	:= TRUE;

				IF NOT interface.cmd.startBrick AND NOT interface.status.commandAck THEN
					gUpperFlapInterface.cmd.start 				:= TRUE;
					interface.status.ready 						:= FALSE;
					interface.status.request					:= FALSE;
					interface.status.commandAck					:= TRUE;
				END_IF
			END_IF

			IF interface.status.commandAck AND (NOT interface.cmd.startBrickOK AND NOT interface.cmd.startBrickNOK AND NOT interface.cmd.startBrick) THEN
				interface.status.commandAck := FALSE;
			END_IF

			CASE em.substate OF
				0:

					IF NOT interface.status.request AND NOT gCapconInterface.status.wingDosing  THEN
						em.substate := 10;
					END_IF

				10:

					em.description := 'waiting for upper flap to be request';

					IF gUpperFlapInterface.status.request  THEN
						interface.status.request 	:= TRUE;
						em.substate 			:= 20;
					END_IF

				20:
					em.description := 'Wait for upperFlap request false';

					IF NOT gUpperFlapInterface.status.request THEN
						em.substate := 0;
					END_IF

			END_CASE

			(**** Manuel mode ****)
			testing;

			this.CycleTimeCalc_0.Enable := em.status.parent.state = STATE_EXECUTE;
			this.CycleTimeCalc_0.MiddleFlapReady := gMiddleFlapInterface.status.ready;
			this.CycleTimeCalc_0.UpperFlapReady := gUpperFlapInterface.status.ready;
			this.CycleTimeCalc_0.Stop := gMiddleFlapInterface.cmd.updateStatistics AND gMiddleFlapInterface.parameter.brickStatus = BRICK_STATUS_OK;
			this.CycleTimeCalc_0();

			this.hmi.cycleTime := this.CycleTimeCalc_0.CycleTime;
			this.hmi.cycleTimeTmu := this.CycleTimeCalc_0.TMU;

			gMiddleFlapInterface.cmd.updateStatistics := FALSE;

			CASE this.waitTimeState OF
				0:
					IF interface.cmd.startBrickOK OR interface.cmd.startBrickNOK THEN
						this.utilityBufferActive := TRUE;	// only start buffer after first element fall through capcon.
						this.waitTimeState := 10;
					END_IF
				10:
					this.waitTime :=this. waitTime + em.status.cycleTime;
					IF gMiddleFlapInterface.status.ready  THEN
						this.waitTimeState := 0;
					END_IF
			END_CASE

			this.waitingTimeUtilisation := this.waitingTimeUtilisation + em.status.cycleTime;
			IF 1000000 < this.waitingTimeUtilisation AND this.utilityBufferActive THEN // wait 1 sec and wait for first element to fall through capcon.
				IF this.waitingTimeBuffer[0] = 0 THEN
					FOR j := 0 TO 59 DO
						this.waitingTimeBuffer[j] := UDINT_TO_REAL(this.waitTime);	// if buffer is new fill the whole buffer with the first result
					END_FOR
				ELSE
					this.waitingTimeBuffer[this.waitingTimeIdx] := UDINT_TO_REAL(this.waitTime);
				END_IF
				this.waitingTimeIdx := (this.waitingTimeIdx+1) MOD 60; // 60 samples in ring buffer
				this.waitTime := 0;
				this.waitingTimeUtilisation := 0;
				this.hmi.waitTimeUtilisation	:= 0;
				FOR j := 0 TO 59 DO
					this.hmi.waitTimeUtilisation := this.hmi.waitTimeUtilisation + this.waitingTimeBuffer[j];
				END_FOR
				this.hmi.waitTimeUtilisation := 100-(this.hmi.waitTimeUtilisation/60000000)*100;
			END_IF

			// Command from main that we should empty now.
			IF gWingInterface.cmd.emptyStart THEN
				gWingInterface.cmd.emptyStart := FALSE;
				em.cmd.complete := TRUE;
			END_IF

			gBottomFlapInterface.parameter.shaftMode 	:= SEL(interface.cmd.shaftModeEmpty, SHAFT_MODE_NORMAL, SHAFT_MODE_EMPTY);	// set shaft mode for bottom flap
			IF interface.cmd.shaftModeEmpty AND NOT this.oldEmptyMode THEN
				// Rising edge on empty mode.
				gBottomFlapInterface.cmd.waitModeChange := TRUE;
			END_IF
			this.oldEmptyMode := interface.cmd.shaftModeEmpty;

			em.cmd.sc									:= TRUE;

		STATE_COMPLETE:
			em.description 				:= 'Emptying machine';

			interface.status.request					:= TRUE;
			IF interface.cmd.confirmEmpty OR gMainInterface.status.state <> STATE_COMPLETING THEN
				interface.cmd.confirmEmpty := FALSE;
				interface.status.commandAck := FALSE;
				em.cmd.stop := TRUE;
			END_IF
			em.cmd.sc := TRUE;

		STATE_STOPPING,STATE_ABORTING,STATE_SUSPENDING:
			em.description 				:= 'clear wing ready signal';
			interface.status.ready 		:= FALSE;
			interface.status.startTestSequence := FALSE;
			interface.status.commandAck := FALSE;
			this.test.startTestSequence := this.test.runUpperFlapContinuously := this.test.runMiddleFlapContinuously := this.test.runBottomFlapContinuously := FALSE;
			em.cmd.sc					:= TRUE;

		STATE_ABORTED:
			em.description := 'waiting for achknowledge comand';
			IF  NOT MpAlarmXCheckReaction(mpAlarmXCore,'abortWing') THEN
				em.cmd.sc 		:= TRUE;
			END_IF

		STATE_CLEARING:
			em.description := 'reset and clear alarms';
			brsmemset(ADR(this.alarm), 0, SIZEOF(this.alarm));
			em.cmd.sc := TRUE;

		STATE_SUSPENDED:

			IF  NOT MpAlarmXCheckReaction(mpAlarmXCore,'abortWing') THEN
				em.cmd.start := TRUE;
				em.cmd.sc := TRUE;
			END_IF

		ELSE
			em.cmd.sc := TRUE;

	END_CASE

END_ACTION
```

#### alarm.st
```iecst
ACTION alarm:

END_ACTION
```

#### wing.st - Init, cyclic, exit code
```iecst
PROGRAM _INIT

	em.setup.name 			:= 'wing';
	em.setup.reactTo 		:= BRDK_EM_REACT_TO_ALL;

	em.setup.lastActivated	:= TRUE;

	// gets the task name and setup names for config and receipe types
	ST_name(0,ADR(this.configName),0);
	brdkStrCpy(ADR(this.recipeName),ADR(this.configName));
	brdkStrCpy(ADR(this.recipeNameCurrent),ADR(this.configName));
	brdkStrCat(ADR(this.configName),ADR(':this.hmi.config'));
	brdkStrCat(ADR(this.recipeName),ADR(':this.hmi.recipe'));
	brdkStrCat(ADR(this.recipeNameCurrent),ADR(':this.hmi.recipeCurrent'));

	setupPointers;
	// Init recipe/config
	config.cassetteDetectTime := 25000;
	config.cassetteReleaseTime := 25000;
	config.readyDelay := 230000;
	config.emptySmallItemsTime := 2000000;
	config.transmissionDelay := 10000;
	config.simCassette := FALSE;
	config.simNeighbour := FALSE;
	config.addFallTimeBottom := 70000;
	// recipe wing timings:
	recipe.flapOpenTimeMiddle.normal := 210000;
	recipe.flapOpenTimeMiddle.Long := 560000;
	recipe.flapOpenTimeUpper.normal := 130000;
	recipe.flapOpenTimeUpper.Long := 360000;
	recipe.flapOpenTimeBottom.normal := 60000;
	recipe.flapOpenTimeBottom.Long := 360000;
	recipe.fallTimeUM := 110000;
	recipe.fallTimeBottom := 260000;
	recipe.longBrick := FALSE;
	recipe.fallTimeBottomLong := 460000;
	recipe.fallTimeBottomNormal := 260000;

END_PROGRAM

PROGRAM _CYCLIC

	setupPointers;

	gWingInterface.parameter.simulation := config.simWing;

	gWingInterface.status.wingEmpty		:= gUpperFlapInterface.status.ready AND gMiddleFlapInterface.status.ready AND gBottomFlapInterface.status.ready1;

	// select if the time is for a short or long brick
	IF recipe.longBrick THEN
		gUpperFlapInterface.parameter.openTime 	:= recipe.flapOpenTimeUpper.Long;
		gMiddleFlapInterface.parameter.openTime := recipe.flapOpenTimeMiddle.Long;
		gBottomFlapInterface.parameter.openTime := recipe.flapOpenTimeBottom.Long;
		gBottomFlapInterface.parameter.fallTime	:= recipe.fallTimeBottomLong;
		config.mediumFlaps := FALSE; // medium not allowed while having long.
	ELSIF config.mediumFlaps THEN
		gUpperFlapInterface.parameter.openTime 	:= recipe.flapOpenTimeUpper.normal;
		gMiddleFlapInterface.parameter.openTime := recipe.flapOpenTimeMiddle.normal;
		gBottomFlapInterface.parameter.openTime := recipe.flapOpenTimeBottom.normal;
		gBottomFlapInterface.parameter.fallTime	:= recipe.fallTimeBottomNormal+config.addFallTimeBottom;
	ELSE
		gUpperFlapInterface.parameter.openTime 	:= recipe.flapOpenTimeUpper.normal;
		gMiddleFlapInterface.parameter.openTime := recipe.flapOpenTimeMiddle.normal;
		gBottomFlapInterface.parameter.openTime := recipe.flapOpenTimeBottom.normal;
		gBottomFlapInterface.parameter.fallTime	:= recipe.fallTimeBottomNormal;
	END_IF

	// set flap times
	gUpperFlapInterface.parameter.flapTime 	:= config.flapMoveTime;
	gMiddleFlapInterface.parameter.flapTime := config.flapMoveTime;
	gBottomFlapInterface.parameter.flapTime := config.flapBottomMoveTime;

	gMiddleFlapInterface.parameter.emptySmallItemsTime 	:= config.emptySmallItemsTime;
	gMiddleFlapInterface.cmd.smallBrick					:= gVibratorInterface[0].status.machineType=0; // Only empty small bricks if it's a small CM20.
	gMiddleFlapInterface.parameter.fallTime				:= recipe.fallTimeUM;

	// Transmission delay.
	gBottomFlapInterface.parameter.transmissionDelay := config.transmissionDelay;
	gBottomFlapInterface.parameter.cassetteStartDelay := config.readyDelay;

	// set pther timers
	gCassetteInterface.parameter.cassetteDetectTime := config.cassetteDetectTime;
	gCassetteInterface.parameter.releaseTime 		:= config.cassetteReleaseTime;
	gWingInterface.status.simCassette := this.hmi.config.simCassette OR gMainInterface.status.simulation;
	gWingInterface.status.simNeighbour := this.hmi.config.simNeighbour;

	interface.status.timeTOF_cassetteSignals := config.timeTOF_cassetteSignals;

	//Normally belt will run when upperFlap close command = TRUE. If this is greater than 0 we will wait that time before telling belt to run.
	gUpperFlapInterface.parameter.startBeltWaitTime := config.startBeltWaitTime;

	CASE em.mode OF
		MODE_PRODUCING,MODE_EMPTY: producing;
		MODE_MANUAL: testing;	// mode for testing flaps manually.
		ELSE em.cmd.sc := TRUE;
	END_CASE

	em();

	alarm;

	this.hw.do_active := TRUE;

	// copy the recipe data
	CASE interface.cmd.copyRecipe OF

		COPY_RECIPE_NEXT_TO_WORKING:
			this.hmi.recipe 			:= this.hmi.recipeCurrent;
			gRecipe.cmd.save 			:= TRUE;
			config.mediumFlaps 			:= FALSE;
			interface.cmd.copyRecipe 	:= COPY_RECIPE_NONE;

		COPY_RECIPE_SANDBOX_TO_NEXT:
			interface.cmd.copyRecipe 	:= COPY_RECIPE_NONE;

	END_CASE

	IF gRecipe.status.doCheckForChanges AND NOT this.oldCheckChangesRecipe THEN
		this.MpRecipeRegPar_Recipe.Enable := TRUE;
		this.MpRecipeRegPar_RecipeCurrent.Enable := TRUE;

		IF gRecipe.status.loaded AND NOT this.oldLoadedRecipe THEN
			// Initial program load. Set old=new to avoid saving just after a load (makes no sense)
			this.recipeOld := this.hmi.recipe;
		END_IF
		this.oldLoadedRecipe := gRecipe.status.loaded;

		IF NOT gRecipe.cmd.save AND gRecipe.status.loaded AND (brsmemcmp(ADR(this.hmi.recipe),ADR(this.recipeOld),SIZEOF(this.recipeOld)) <> 0) THEN
			gRecipe.cmd.save := TRUE;
			this.recipeOld := this.hmi.recipe;
		END_IF

	END_IF
	this.MpRecipeRegPar_Recipe(MpLink := ADR(mpRecipe), PVName := ADR(this.recipeName), Category := ADR('recipe'));
	this.MpRecipeRegPar_RecipeCurrent(MpLink := ADR(mpRecipeCurrent), PVName := ADR(this.recipeNameCurrent), Category := ADR('recipeCurrent'));
	this.oldCheckChangesRecipe := gRecipe.status.doCheckForChanges;

	IF gConfig.status.doCheckForChanges AND NOT this.oldCheckChangesConfig THEN
		this.MpRecipeRegPar_Config.Enable := TRUE;

		IF gConfig.status.loaded AND NOT this.oldLoaded THEN
			// Initial program load. Set old=new to avoid saving just after a load (makes no sense)
			this.configOld := this.hmi.config;
		END_IF
		this.oldLoaded := gConfig.status.loaded;

		IF NOT gConfig.cmd.save AND gConfig.status.loaded AND (brsmemcmp(ADR(this.hmi.config),ADR(this.configOld),SIZEOF(this.configOld)) <> 0) THEN
			gConfig.cmd.save := TRUE;
			this.configOld := this.hmi.config;
		END_IF

	END_IF
	this.MpRecipeRegPar_Config(MpLink := ADR(mpRecipe), PVName := ADR(this.configName), Category := ADR('config'));
	this.oldCheckChangesConfig := gConfig.status.doCheckForChanges;

	IF gConfig.status.factoryReset[4] THEN // Both cassette/wing
		gConfig.status.factoryReset[4] := FALSE;
		// Factory reset all parameters:
		config.cassetteDetectTime := 25000;
		config.cassetteReleaseTime := 25000;
		config.readyDelay := 230000;
		config.emptySmallItemsTime := 2000000;
		config.transmissionDelay := 10000;
		config.simCassette := FALSE;
		config.simNeighbour := FALSE;
		config.addFallTimeBottom := 70000;
		// recipe wing timings:
		recipe.flapOpenTimeMiddle.normal := 210000;
		recipe.flapOpenTimeMiddle.Long := 560000;
		recipe.flapOpenTimeUpper.normal := 130000;
		recipe.flapOpenTimeUpper.Long := 360000;
		recipe.flapOpenTimeBottom.normal := 60000;
		recipe.flapOpenTimeBottom.Long := 360000;
		recipe.fallTimeUM := 110000;
		recipe.fallTimeBottom := 260000;
		recipe.longBrick := FALSE;
		recipe.fallTimeBottomLong := 460000;
		recipe.fallTimeBottomNormal := 260000;

	END_IF

END_PROGRAM

PROGRAM _EXIT

	this.MpRecipeRegPar_Recipe(Enable := FALSE);
	this.MpRecipeRegPar_Config(Enable := FALSE);
	this.MpRecipeRegPar_RecipeCurrent(Enable := FALSE);

END_PROGRAM
```

#### testing.st
```iecst
ACTION testing:

	CASE this.test.state OF

		0:
			IF this.test.startTestSequence THEN
				interface.status.startTestSequence := TRUE;
				gUpperFlapInterface.cmd.runFlapContinuously := this.test.runUpperFlapContinuously := FALSE;
				gMiddleFlapInterface.cmd.runFlapContinuously := this.test.runMiddleFlapContinuously := FALSE;
				gBottomFlapInterface.cmd.runFlapContinuously := this.test.runBottomFlapContinuously := FALSE;
				gUpperFlapInterface.cmd.manuelMode := gMiddleFlapInterface.cmd.manuelMode := gBottomFlapInterface.cmd.manuelMode := TRUE;
				this.test.state := 20;
			ELSIF this.test.runUpperFlapContinuously OR this.test.runMiddleFlapContinuously OR this.test.runBottomFlapContinuously THEN
				this.test.state := 10;
			ELSE
				gUpperFlapInterface.cmd.manuelMode := gMiddleFlapInterface.cmd.manuelMode := gBottomFlapInterface.cmd.manuelMode := interface.status.startTestSequence := FALSE;
			END_IF

		(**** Actuate flaps continously if prompted from hmi. ****)

		10:
			gUpperFlapInterface.cmd.runFlapContinuously := gUpperFlapInterface.cmd.manuelMode := this.test.runUpperFlapContinuously;
			gMiddleFlapInterface.cmd.runFlapContinuously := gMiddleFlapInterface.cmd.manuelMode := this.test.runMiddleFlapContinuously;
			gBottomFlapInterface.cmd.runFlapContinuously := gBottomFlapInterface.cmd.manuelMode := this.test.runBottomFlapContinuously;

			IF (NOT this.test.runUpperFlapContinuously AND NOT this.test.runMiddleFlapContinuously AND NOT this.test.runBottomFlapContinuously) OR this.test.startTestSequence THEN
				gUpperFlapInterface.cmd.runFlapContinuously := this.test.runUpperFlapContinuously := FALSE;
				gMiddleFlapInterface.cmd.runFlapContinuously := this.test.runMiddleFlapContinuously := FALSE;
				gBottomFlapInterface.cmd.runFlapContinuously := this.test.runBottomFlapContinuously := FALSE;
				this.test.state := 0;
			END_IF

		(**** Start flap sequence ****)

		20:

			IF NOT this.test.startTestSequence THEN	// test stopped
				gUpperFlapInterface.cmd.runFlapContinuously := gUpperFlapInterface.cmd.open := FALSE;
				gMiddleFlapInterface.cmd.runFlapContinuously := gMiddleFlapInterface.cmd.open := FALSE;
				gBottomFlapInterface.cmd.runFlapContinuously := gBottomFlapInterface.cmd.open := FALSE;
				interface.status.startTestSequence := FALSE;
				this.test.state := 0;
			ELSE
				// Signal flaps to open in a sequence.
				gUpperFlapInterface.cmd.open := TRUE;
				this.test.state := 30;
			END_IF

		30:
			em.description := 'Wait for upper flap to open/close';

			IF NOT this.test.startTestSequence THEN
				gUpperFlapInterface.cmd.open := FALSE;
				interface.status.startTestSequence := FALSE;
				this.test.state := 0;
			ELSIF NOT gUpperFlapInterface.cmd.open THEN // means that it has been open and closed.
				gMiddleFlapInterface.cmd.open := TRUE;
				this.test.state := 40;
			END_IF

		40:
			em.description := 'Wait for middle flap to open/close';

			IF NOT this.test.startTestSequence THEN
				gMiddleFlapInterface.cmd.open := FALSE;
				interface.status.startTestSequence := FALSE;
				this.test.state := 0;
			ELSIF NOT gMiddleFlapInterface.cmd.open THEN
				gBottomFlapInterface.cmd.open := TRUE;
				this.test.state := 50;
			END_IF

		50:
			em.description := 'Wait for bottom flap to open/close';

			IF NOT this.test.startTestSequence THEN
				gBottomFlapInterface.cmd.open := FALSE;
				interface.status.startTestSequence := FALSE;
				this.test.state := 0;
			ELSIF NOT gBottomFlapInterface.cmd.open THEN
				this.test.state := 20;
			END_IF

	END_CASE

END_ACTION
```

#### setupPointers.st
```iecst
ACTION setupPointers:
	recipe ACCESS ADR(this.hmi.recipe);
	config ACCESS ADR(this.hmi.config);
	interface ACCESS ADR(gWingInterface);
END_ACTION
```

#### local.typ - Local data types
```iecst
TYPE
	hmi_typ : 	STRUCT
		upperAccept : BOOL;
		upperReject : BOOL;
		upperClosed : BOOL;
		upperChangeOverToClosed : BOOL;
		upperChangeOverToOpened : BOOL;
		middleAccept : BOOL;
		middleReject : BOOL;
		middleClosed : BOOL;
		middleChangeOverToClosed : BOOL;
		middleChangeOverToOpened : BOOL;
		bottomAccept : BOOL;
		bottomReject : BOOL;
		bottomOpened : BOOL;
		bottomClosed : BOOL;
		bottomChangeOverToClosed : BOOL;
		bottomChangeOverToOpened : BOOL;
		middleNeighbourAccept : BOOL;
		bottomNeighbourAccept : BOOL;
		bottomNeighbourOpened : BOOL;
		bottomNeighbourClosed : BOOL;
		bottomNeighbourChangeOverToClose : BOOL;
		bottomNeighbourChangeOverToOpen : BOOL;
		cmd : hmi_cmd_typ;
		config : config_wing_typ;
		recipe : recipe_wing_typ;
		cycleTime : REAL;
		cycleTimeTmu : REAL;
		waitTimeUtilisation : REAL;
		recipeCurrent : recipe_wing_typ;
		addFallTimeMs : UDINT;
	END_STRUCT;
	hmi_cmd_typ : 	STRUCT
		rejectAll : SINT;
	END_STRUCT;
	local_typ : 	STRUCT
		hw : local_hw_typ;
		alarm : local_alarm_typ;
		MpRecipeRegPar_Config : MpRecipeRegPar;
		MpRecipeRegPar_Recipe : MpRecipeRegPar;
		MpRecipeRegPar_RecipeCurrent : MpRecipeRegPar;
		brdkPVLocalVariable_0 : brdkPVLocalVariable;
		time : local_time_typ;
		hmi : hmi_typ;
		configName : STRING[80];
		recipeName : STRING[80];
		recipeNameCurrent : STRING[80];
		configOld : config_wing_typ;
		recipeOld : recipe_wing_typ;
		middelBrickStatusTmp : gFlap_brick_status_typ;
		start : BOOL;
		upperReadyOld : BOOL;
		middleFlapStartOld : BOOL;
		cycleTime : UDINT;
		cycleTimeIdx : USINT;
		cycleTimes : ARRAY[0..9]OF REAL;
		cycleTimesTmu : ARRAY[0..9]OF REAL;
		waitingTimeUtilisation : UDINT;
		waitingTimeIdx : USINT;
		waitingTimeBuffer : ARRAY[0..59]OF REAL;
		waitTime : UDINT;
		waitTimeState : USINT;
		machineStartOld : BOOL;
		utilityBufferActive : BOOL; (*true when utility buffer is active.*)
		blockCycleTime : BOOL; (*if true we don't meassure cycle time*)
		oldEmptyMode : BOOL;
		stateStatisctics : USINT;
		CycleTimeCalc_0 : CycleTimeCalc;
		test : local_test_typ;
		oldCheckChangesConfig : BOOL;
		oldCheckChangesRecipe : BOOL;
		oldLoaded : BOOL;
		oldLoadedRecipe : BOOL;
	END_STRUCT;
	local_test_typ : 	STRUCT
		startTestSequence : BOOL;
		runUpperFlapContinuously : BOOL;
		runMiddleFlapContinuously : BOOL;
		runBottomFlapContinuously : BOOL;
		state : USINT;
	END_STRUCT;
	flap_ctrl_typ : 	STRUCT
		state : USINT;
		description : STRING[65];
		ready : BOOL;
		accept : BOOL;
		reject : BOOL;
		fall : BOOL;
		fallTimeLeft : REAL;
	END_STRUCT;
	local_hw_typ : 	STRUCT
		do_active : BOOL; (*Signal name: DO_WU_NCON
PJ95: WU_S
Connector: DO.18
Description: Signal to neighbour CM. �1� means CM is connected and active.*)
		wu_error : ARRAY[0..1]OF BOOL; (*WU_error*)
	END_STRUCT;
	config_wing_typ : 	STRUCT
		readyDelay : UDINT := 0; (*Delay before the ready seignal is activated.*)
		flapMoveTime : UDINT := 800000; (*Time that the flap is to move.*)
		flapBottomMoveTime : UDINT := 800000; (*Time that the bottom flap is to move.*)
		cassetteDetectTime : UDINT := 20000; (*Time that the cassette ready signal need to be low*)
		cassetteReleaseTime : UDINT := 20000; (*Cassette release time*)
		simCassette : BOOL := FALSE; (*Simulate the cassette*)
		simNeighbour : BOOL := FALSE; (*Simulate the neigbour*)
		emptySmallItemsTime : UDINT := 2000000; (*Time middle flap is closed before letting out  smll itmes for empty.*)
		transmissionDelay : UDINT := 10000;
		startBeltWaitTime : UDINT := 0; (*Normally belt will run when upperFlap close command = TRUE. If this is greater than 0 we will wait that time before telling belt to run.*)
		simWing : BOOL := FALSE;
		timeTOF_cassetteSignals : TIME := T#250ms;
		mediumFlaps : BOOL; (*Required for special element like rubber tires. They need to run a bit slower flaps but "long" flaps reduce cycle time too much*)
		addFallTimeBottom : UDINT := 70000;
	END_STRUCT;
	recipe_wing_typ : 	STRUCT
		flapOpenTimeMiddle : recipe_flap_open_time_typ; (*Time that the flaps stays open for normal bricks.*)
		flapOpenTimeUpper : recipe_flap_open_time_typ; (*Time that the flaps stays open for normal bricks.*)
		flapOpenTimeBottom : recipe_flap_open_time_typ;
		fallTimeUM : UDINT := 100000;
		fallTimeBottom : UDINT := 100000; (*Time to fall from middle to bottom flap*)
		longBrick : BOOL;
		fallTimeBottomLong : UDINT := 460000;
		fallTimeBottomNormal : UDINT := 260000;
	END_STRUCT;
	neighbourState_typ :
		(
		NEIGHBOUR_NOT_ACTIVE := 0,
		NEIGHBOUR_ACTIVE := 1
		);
	local_alarm_typ : 	STRUCT
		dummy : USINT;
	END_STRUCT;
	local_time_typ : 	STRUCT
		elapsed : UDINT;
		maximum : UDINT;
	END_STRUCT;
	recipe_flap_open_time_typ : 	STRUCT
		normal : UDINT := 110000;
		Long : UDINT := 360000;
	END_STRUCT;
END_TYPE
```

#### local.var - Local variables
```iecst
VAR
	j : USINT;
	this : {REDUND_UNREPLICABLE} local_typ;
	em : {REDUND_UNREPLICABLE} brdkEM;
	recipe : REFERENCE TO recipe_wing_typ;
	config : REFERENCE TO config_wing_typ;
	interface : REFERENCE TO gWingInterface_typ;
END_VAR
```

#### LocalFunctions.fun
```iecst
{REDUND_ERROR} FUNCTION_BLOCK CycleTimeCalc (*TODO: Add your comment here*) (*$GROUP=User,$CAT=User,$GROUPICON=User.png,$CATICON=User.png*)
	VAR_INPUT
		Enable : {REDUND_UNREPLICABLE} BOOL;
		UpperFlapReady : BOOL;
		MiddleFlapReady : BOOL;
		Stop : BOOL;
	END_VAR
	VAR_OUTPUT
		Ready : BOOL;
		CycleTime : REAL;
		TMU : REAL;
	END_VAR
	VAR
		startTime1 : TIME;
		startTime2 : TIME;
		elapsed : TIME;
		tmu : REAL;
		cycleTime : REAL;
		cycleTimeArr : ARRAY[0..9] OF REAL;
		cycleTimeArrFull : BOOL;
		cycleTimeArrIdx : USINT;
		state : UDINT;
		i : UDINT;
		_stop : BOOL;
	END_VAR
END_FUNCTION_BLOCK
```

#### LocalFunctions.st
```iecst
(* Calculates cycle time for CM20 *)
FUNCTION_BLOCK CycleTimeCalc

	IF Enable THEN
		Ready := TRUE;

		IF Stop AND NOT _stop THEN
			_stop := TRUE;
		END_IF

		CASE state OF
			0: // Waiting for Upper or Middle to be ready
				IF MiddleFlapReady OR UpperFlapReady THEN
					IF startTime1 = T#0ms THEN
						startTime1 := clock_ms();
					END_IF
					elapsed := 0;
					state := 10;
				END_IF
			10:
				IF NOT UpperFlapReady AND NOT MiddleFlapReady THEN
					elapsed := clock_ms()-startTime1;
					state := 20;
				ELSIF NOT UpperFlapReady THEN
					state := 30;
				END_IF
			20:
				IF MiddleFlapReady THEN
					startTime1 := clock_ms();
					state := 30;
				END_IF
			30:
				IF UpperFlapReady THEN
					startTime2 := clock_ms();
					state := 40;
				ELSIF _stop THEN
					_stop := FALSE;
					elapsed := elapsed + (clock_ms()-startTime1);
					cycleTimeArr[cycleTimeArrIdx] := TIME_TO_REAL(elapsed)/1000.0;
					cycleTimeArrFull := SEL(cycleTimeArrIdx = 9, cycleTimeArrFull, TRUE);
					cycleTimeArrIdx := SEL(cycleTimeArrIdx = 9, cycleTimeArrIdx + 1, 0);
					cycleTime := 0;
					IF cycleTimeArrIdx > 0 OR cycleTimeArrFull THEN
						FOR i:=0 TO SEL(cycleTimeArrFull, cycleTimeArrIdx-1, 9) DO
							cycleTime := cycleTime + cycleTimeArr[i]/SEL(cycleTimeArrFull, USINT_TO_REAL(cycleTimeArrIdx), 10.0);
						END_FOR
						CycleTime := 60.0/cycleTime;
						tmu := 0;
						FOR i:=0 TO SEL(cycleTimeArrFull, cycleTimeArrIdx-1, 9) DO
							tmu := tmu + cycleTimeArr[i]/360.0;
						END_FOR
						TMU := tmu;
					END_IF
					state := 0;
				END_IF
			40:
				IF _stop THEN
					_stop := FALSE;
					elapsed := elapsed + (clock_ms()-startTime1);
					cycleTimeArr[cycleTimeArrIdx] := TIME_TO_REAL(elapsed)/1000.0;
					cycleTimeArrFull := SEL(cycleTimeArrIdx = 9, cycleTimeArrFull, TRUE);
					cycleTimeArrIdx := SEL(cycleTimeArrIdx = 9, cycleTimeArrIdx + 1, 0);
					cycleTime := 0;
					IF cycleTimeArrIdx > 0 OR cycleTimeArrFull THEN
						FOR i:=0 TO SEL(cycleTimeArrFull, cycleTimeArrIdx-1, 9) DO
							cycleTime := cycleTime + cycleTimeArr[i]/SEL(cycleTimeArrFull, USINT_TO_REAL(cycleTimeArrIdx), 10.0);
						END_FOR
						CycleTime := 60.0/cycleTime;
						tmu := cycleTime/0.0360;
						TMU := tmu;
					END_IF
					startTime1 := startTime2;
					startTime2 := T#0ms;
					state := 0;
				END_IF
		END_CASE

	ELSIF Ready THEN
		Ready := FALSE;
		brsmemset(ADR(cycleTimeArr), 0, SIZEOF(cycleTimeArr));
		cycleTimeArrFull := FALSE;
		cycleTimeArrIdx := 0;
		CycleTime := 0;
		TMU := 0;
		startTime1 := T#0ms;
		startTime2 := T#0ms;
	END_IF

END_FUNCTION_BLOCK
```

### wingGlobal.typ
```iecst
TYPE
	gWingInterface_typ : 	STRUCT
		cmd : gWingInterface_cmd_typ;
		parameter : gWingInterface_parameter_typ;
		status : gWingInterface_status_typ;
	END_STRUCT;
	gWingInterface_cmd_typ : 	STRUCT
		startBrickNOK : BOOL; (*Start wing with NOK brick.*)
		startBrickOK : BOOL; (*Start wing with OK brick.*)
		emptyStart : BOOL;
		emptyStop : BOOL;
		dosing : BOOL;
		shaftModeEmpty : BOOL;
		machineStart : BOOL;
		startManuelMode : BOOL;
		changeMode : BOOL; (*signal from wing -> main to change mode*)
		copyRecipe : copy_recipe_command_typ;
		rejectNextBatch : BOOL; (*Used if we have an aftercount to reject the next batch as well. We both need to reject upper/middle in case of afterCount*)
		disableOptimization : BOOL; (*Used to disable wing flap optimization (FOR TEST)*)
		startBrick : BOOL;
		confirmEmpty : BOOL;
	END_STRUCT;
	gWingInterface_status_typ : 	STRUCT
		neighbourActive : BOOL;
		ready : BOOL;
		simCassette : BOOL;
		simNeighbour : BOOL;
		request : BOOL;
		commandAck : BOOL;
		startTestSequence : BOOL;
		wingEmpty : BOOL;
		stepperWUConnected : BOOL;
		timeTOF_cassetteSignals : TIME;
	END_STRUCT;
	gWingInterface_parameter_typ : 	STRUCT
		simulation : BOOL;
	END_STRUCT;
	local_time_typ : 	STRUCT
		elapsed : UDINT;
		maximum : UDINT;
	END_STRUCT;
	gFlap_brick_status_typ :
		(
		BRICK_STATUS_NOK := 0, (*Reject brick(s)*)
		BRICK_STATUS_OK := 1, (*Good brick(s)*)
		BRICK_STATUS_REJECT_ALL := 2, (*Reject all*)
		BRICK_STATUS_EMPTY := 3, (*Empty mode*)
		BRICK_STATUS_EMPTY_SMALL_ITEMS := 4, (*Empty small items*)
		BRICK_STATUS_EMPTY_END := 5, (*Empty ends*)
		BRICK_STATUS_DOSING := 6, (*Dosing*)
		BRICK_STATUS_DOSING_AND_EMPTY := 7 (*Dosing and empty*)
		);
END_TYPE
```

### wingGlobal.var
```iecst
VAR
	gWingInterface : gWingInterface_typ;
END_VAR
```

### Program Logical/modules/main/wing/upperFlap/upperFlap (IEC)

#### producing.st
```iecst
ACTION producing:

	CASE em.state OF

		STATE_STOPPED:

			interface.status.active := TRUE; // need to tell wing when we are active. (otherwise wing start too fast and this task is stuck in STATE_ACTIVATING doing boot)

			interface.status.ready 	:= FALSE;
			interface.status.request := FALSE;

			em.cmd.sc 				:= TRUE;

		STATE_RESETTING:

			em.cmd.sc := TRUE;

		STATE_STARTING:

			interface.status.request := TRUE; // request new brick
			interface.status.ready 	:= TRUE;
			interface.cmd.start		:= FALSE;
			em.cmd.sc 				:= TRUE;

		STATE_EXECUTE:

			CASE em.substate OF

				0:	// G010 (Initialisation)
					em.cmd.sc := TRUE;
					interface.status.ready	:= TRUE; // only ready if not about to reject due to aftercount.;

					em.description := 'waiting for start command';

//					IF this.afterCount THEN
//
//						IF (interface.status.request AND interface.cmd.start) OR NOT interface.status.request THEN
//							interface.cmd.start 		:= FALSE;
//							//this.afterCount := FALSE;
//							interface.status.request	 := FALSE;
//							interface.status.ready 		:= FALSE;
//							em.substate := 20;
//						END_IF
//
					IF interface.cmd.start THEN
						interface.cmd.start 		:= FALSE;
						this.waitingTime.current	:= 0;
						interface.status.request	 := FALSE;
						interface.status.ready 		:= FALSE;

						this.lastUpperFlapCycleTime := this.upperFlapCycleTime;

						em.substate := 20;
					ELSIF interface.cmd.manuelMode THEN
						em.substate := 1000;
					END_IF

				20: // G020 (Shaft Start)
					em.description := 'waiting for middle flap to be ready';
					this.waitingTime.current := this.waitingTime.current + em.status.cycleTime;

					IF gCapconInterface.status.brickPresent AND interface.cmd.brickStatusReady AND gCapconInterface.parameter.capconMode <> 2 THEN // don't look on aftercount from capcon if capconMode=OFF
						this.rejectNext := TRUE;
					END_IF

					IF gMiddleFlapInterface.status.ready THEN
						this.flap.open := TRUE;
						this.cycleTimeTheoretical := 0;
						this.upperFlapCycleTime := 0;
						em.substate := 50;
						em.cmd.sc := FALSE;
					END_IF

				50: // G050 (Open FU)
					em.description 				:= 'waiting for flap to be open';

					IF gCapconInterface.status.brickPresent AND interface.cmd.brickStatusReady AND gCapconInterface.parameter.capconMode <> 2 THEN // don't look on aftercount from capcon if capconMode=OFF
						this.rejectNext := TRUE;
					END_IF

					IF this.flap.error THEN
						this.alarm.openTooLong.active := TRUE;
						this.previousState := em.substate;
						em.substate := 700; // Error in execute
					ELSIF this.flap.position = FLAP_OPEN THEN
						this.time.elapsed		:= 0;
						this.time.maximum		:= interface.parameter.openTime;
						em.substate 			:= 55;
					END_IF

				55:
					em.description 		:= 'waiting for open time';

					IF gCapconInterface.status.brickPresent AND interface.cmd.brickStatusReady AND gCapconInterface.parameter.capconMode <> 2 THEN // don't look on aftercount from capcon if capconMode=OFF
						this.rejectNext := TRUE;
					END_IF

					this.time.elapsed	:= this.time.elapsed + em.status.cycleTime;

					IF this.time.elapsed >= this.time.maximum AND (NOT interface.status.ready OR interface.cmd.brickStatusReady) THEN
						this.flap.close := TRUE;
						interface.status.request := TRUE;	 // if no wait time set true now. Otherwise wait time from config.
						gMiddleFlapInterface.parameter.brickStatus := SEL(this.rejectNext OR this.afterCount , interface.parameter.brickStatus, BRICK_STATUS_NOK);
						this.afterCount := this.rejectNext := FALSE;

						interface.cmd.brickStatusReady := FALSE;
						interface.status.openCloseTime := this.cycleTimeTheoretical;
						this.time.elapsed := 0;
						em.substate	:= 60;
					END_IF

				60: // G060 (Close FU)
					em.description := 'waiting for after count time';

					this.time.elapsed := this.time.elapsed + em.status.cycleTime;

					IF (gCapconInterface.status.brickPresent OR testAfterCount) AND NOT this.afterCount AND gCapconInterface.parameter.capconMode <> 2 THEN // don't look on aftercount from capcon if capconMode=OFF
						testAfterCount := FALSE;
						this.afterCount := TRUE;
					ELSIF (this.time.elapsed/1000) >= (this.flap.closingTimeAfterChangeover-90) OR this.flap.position = FLAP_CLOSED THEN
						IF this.afterCount AND gCapconInterface.parameter.capconMode <> 2 THEN // don't look on aftercount from capcon if capconMode=OFF
							interface.parameter.brickStatus := BRICK_STATUS_NOK;
							gMiddleFlapInterface.parameter.brickStatus := BRICK_STATUS_NOK;
							//gBeltInterface.cmd.afterCount := TRUE;
						END_IF
						interface.status.lastCycleTime := this.upperFlapCycleTime;

						// Don't calculate reject% if about to do extra motion after afterCount or doing a teach.
						IF NOT this.afterCount AND gCapconInterface.status.teachingDone THEN
							this.errBuffer_0.input := gMiddleFlapInterface.parameter.brickStatus = BRICK_STATUS_OK;
							this.errBuffer_0.pushToBuffer := this.oldTeachingDone;
							this.errBuffer_0();
							this.hmi.errorRate := this.errBuffer_0.errorRate*100;
							interface.status.OKPortions := SEL(gMiddleFlapInterface.parameter.brickStatus = BRICK_STATUS_OK, interface.status.OKPortions, interface.status.OKPortions + 1);
							interface.status.NOKPortions := SEL(gMiddleFlapInterface.parameter.brickStatus = BRICK_STATUS_NOK, interface.status.NOKPortions, interface.status.NOKPortions + 1);
						END_IF
						this.oldTeachingDone := gCapconInterface.status.teachingDone;

						interface.status.countAftercount := SEL(this.afterCount,interface.status.countAftercount,interface.status.countAftercount + 1);

						// If reject all is enabled it should always be a reject
						interface.parameter.brickStatus := SEL(this.hmi.rejectAll,interface.parameter.brickStatus,BRICK_STATUS_NOK);
						gMiddleFlapInterface.parameter.brickStatus := SEL(this.hmi.rejectAll,gMiddleFlapInterface.parameter.brickStatus,BRICK_STATUS_NOK);
						gMiddleFlapInterface.cmd.start := TRUE;

						em.substate := 65;
					END_IF

				65: // G060 (Close FU)
					em.description 		:= 'waiting for flap to be closed';

					IF this.flap.error THEN
						this.alarm.openTooLong.active := TRUE;
						this.previousState := em.substate;
						em.substate := 700; // Error in execute
					ELSIF this.flap.position = FLAP_CLOSED THEN

						IF interface.parameter.brickStatus = BRICK_STATUS_OK THEN
							this.MTFilterMovingAverage_0.Enable := TRUE;
							this.MTFilterMovingAverage_0.In := 60000000.0 / UDINT_TO_REAL(LIMIT(1, this.lastUpperFlapCycleTime, 4000000));
							this.MTFilterMovingAverage_0.WindowLength := 40;
							this.MTFilterMovingAverage_0();

							this.MTFilterMovingAverage_10.Enable := TRUE;
							this.MTFilterMovingAverage_10.In := 60000000.0 / UDINT_TO_REAL(LIMIT(1, this.lastUpperFlapCycleTime, 4000000));
							this.MTFilterMovingAverage_10.WindowLength := 10;
							this.MTFilterMovingAverage_10();

							this.MTFilterMovingAverage_10_TMU.Enable := TRUE;
							this.MTFilterMovingAverage_10_TMU.In := UDINT_TO_REAL(LIMIT(1, this.lastUpperFlapCycleTime, 4000000))/36000;
							this.MTFilterMovingAverage_10_TMU.WindowLength := 10;
							this.MTFilterMovingAverage_10_TMU();
						ELSE
							this.upperFlapCycleTime := this.upperFlapCycleTime + this.lastUpperFlapCycleTime;
						END_IF

						this.flapTest.openTime := this.flap.openTimeAfterChangeover;
						this.flapTest.closingTime := this.flap.closingTimeAfterChangeover;
						this.flapTest.openTimeOK := this.flapTest.openTime >= 210 AND this.flapTest.openTime <= 230;
						this.flapTest.closingTimeOK := this.flapTest.closingTime >= 210 AND this.flapTest.closingTime <= 230;
						em.substate := 0;
					END_IF

					(**** ERROR handling in EXECUTE ****)

				700:
					interface.cmd.runFlapContinuously	:= FALSE;
					interface.cmd.open					:= FALSE;
					interface.cmd.manuelMode			:= FALSE;

					IF NOT this.flap.error THEN
						this.flap.close := TRUE;
						em.substate := 710;
					ELSE
						this.flap.resetError := TRUE;
					END_IF

				710:
					em.description := 'Wait for flap to close - if not still continue. We cant be stuck in "SUSPENDING"';

					IF this.flap.error THEN
						this.time.elapsed := 0;
						em.substate := 720;
					ELSIF this.flap.position = FLAP_CLOSED THEN
						this.time.elapsed := 0;
						em.substate := 720;
					END_IF

				720:
					em.description := 'Wait for alarm acknowledge';

					this.time.elapsed := this.time.elapsed + em.status.cycleTime;

					IF this.time.elapsed >= 500000 THEN //500ms
						this.time.elapsed := 0;
						IF NOT MpAlarmXCheckReaction(mpAlarmXCore,'abortMain') THEN
							em.substate := 730; // "UNSUSPENDING"
						END_IF
					END_IF

				730:
					IF NOT this.flap.error THEN
						brsmemset(ADR(this.alarm), 0, SIZEOF(this.alarm));
						this.alarm.closeTooLong.name := 'upperFlapCloseTooLong';
						this.alarm.openTooLong.name := 'upperFlapOpenTooLong';
						this.flap.close := TRUE;
						em.substate := 740;
					ELSE
						this.flap.resetError := TRUE;
					END_IF

				740:
					em.description := 'Wait for flap to close -> if not go back and try again ';

					IF this.flap.error THEN
						em.substate := 730; // Try again (we MUST close flap before we return)
					ELSIF this.flap.position = FLAP_CLOSED THEN
						em.substate := 750;
					END_IF

				750:
					em.description := 'Recover to "previousState"';

					CASE this.previousState OF

						50: // Error opening
							this.flap.open := TRUE;
							this.cycleTimeTheoretical := 0;
							em.substate := 50;

						65: // Error closing
							this.flap.close := TRUE;
							em.substate := 65;

						1000:
							em.substate := 0;

					END_CASE

					(**** Manuel mode ****)

				1000:
					testing;
					IF this.flap.error THEN
						// Stop testing and go in execute error state.
						this.previousState := em.substate;
						this.test.state := 0;

						em.substate := 700;
					END_IF

			END_CASE

			this.cycleTimeTheoretical := this.cycleTimeTheoretical + em.status.cycleTime;
			IF gMainInterface.status.state = STATE_EXECUTE THEN
				this.upperFlapCycleTime := this.upperFlapCycleTime + em.status.cycleTime;
			END_IF

		STATE_COMPLETING:

			CASE em.substate OF

				0:
					em.description 				:= 'waiting for flap to be open';
					this.flap.open := TRUE;
					IF this.flap.error THEN
						this.alarm.openTooLong.active := TRUE;
						this.previousState := em.substate;
						em.substate := 700;
					ELSIF this.flap.position = FLAP_OPEN THEN
						this.time.elapsed := 0;
						em.substate := 10;
					END_IF
				10:
					em.description 				:= 'waiting for middle flap to be ready';
					em.cmd.sc := gMiddleFlapInterface.status.ready;

					(**** ERROR handling in COMPLETE ****)

				700:
					interface.cmd.runFlapContinuously	:= FALSE;
					interface.cmd.open					:= FALSE;
					interface.cmd.manuelMode			:= FALSE;

					IF NOT this.flap.error THEN
						this.flap.close := TRUE;
						em.substate := 710;
					ELSE
						this.flap.resetError := TRUE;
					END_IF

				710:
					em.description := 'Wait for flap to close - if not still continue. We cant be stuck in "SUSPENDING"';

					IF this.flap.error THEN
						this.time.elapsed := 0;
						em.substate := 720;
					ELSIF this.flap.position = FLAP_CLOSED THEN
						this.time.elapsed := 0;
						em.substate := 720;
					END_IF

				720:
					em.description := 'Wait for alarm acknowledge';

					this.time.elapsed := this.time.elapsed + em.status.cycleTime;

					IF this.time.elapsed >= 500000 THEN //500ms
						this.time.elapsed := 0;
						IF NOT MpAlarmXCheckReaction(mpAlarmXCore,'abortMain') THEN
							em.substate := 730; // "UNSUSPENDING"
						END_IF
					END_IF

				730:
					IF NOT this.flap.error THEN
						brsmemset(ADR(this.alarm), 0, SIZEOF(this.alarm));
						this.alarm.closeTooLong.name := 'upperFlapCloseTooLong';
						this.alarm.openTooLong.name := 'upperFlapOpenTooLong';
						this.flap.close := TRUE;
						em.substate := 740;
					ELSE
						this.flap.resetError := TRUE;
					END_IF

				740:
					em.description := 'Wait for flap to close -> if not go back and try again ';

					IF this.flap.error THEN
						em.substate := 730; // Try again (we MUST close flap before we return)
					ELSIF this.flap.position = FLAP_CLOSED THEN
						em.substate := 750;
					END_IF

				750:
					em.description := 'Recover to "previousState"';

					CASE this.previousState OF

						0: // Error opening
							this.flap.open := TRUE;
							em.substate := 0;

					END_CASE

			END_CASE

		STATE_COMPLETE:

			em.description 				:= 'Emptying machine';
			em.setup.reactTo := BRDK_EM_REACT_TO_ALL;
			interface.status.ready := TRUE;
			interface.status.request := TRUE;
			em.cmd.sc := TRUE;

		STATE_ABORTED, STATE_SUSPENDED:
			em.description := 'waiting for wing to start';
			em.cmd.sc := TRUE;

		STATE_STOPPING, STATE_ABORTING, STATE_SUSPENDING:

			CASE em.substate OF

				0:
					em.description 				:= 'Clear status and close flap';
					interface.status.request := FALSE;
					interface.status.ready 	:= FALSE;
					interface.cmd.start 	:= FALSE;
					interface.cmd.brickStatusReady := FALSE;
					this.hw.do_open := FALSE;
					interface.cmd.runFlapContinuously	:= FALSE;
					interface.cmd.open					:= FALSE;
					interface.cmd.manuelMode			:= FALSE;

					IF NOT this.flap.error THEN
						this.flap.close := TRUE;
						em.substate := 10;
					ELSE
						this.flap.resetError := TRUE;
					END_IF

				10:
					em.description := 'Wait for flap to close';

					IF this.flap.error THEN
						em.substate := 20;
					ELSIF this.flap.position = FLAP_CLOSED THEN
						em.substate := 20;
					END_IF

				20:
					em.cmd.sc := TRUE;

			END_CASE

		STATE_CLEARING, STATE_UNSUSPENDING:
			em.description := 'waiting for flap error reset';

			CASE em.substate OF

				0:
					IF NOT this.flap.error THEN
						brsmemset(ADR(this.alarm), 0, SIZEOF(this.alarm));
						//Alarm texts
						this.alarm.closeTooLong.name := 'upperFlapCloseTooLong';
						this.alarm.openTooLong.name := 'upperFlapOpenTooLong';
						this.flap.close := TRUE;
						em.substate := 10;
					ELSE
						this.flap.resetError := TRUE;
					END_IF

				10:
					em.description := 'Wait for flap to close';

					IF this.flap.error THEN
						em.substate := 0;
					ELSIF this.flap.position = FLAP_CLOSED  THEN
						interface.status.request := TRUE;
						em.substate := 20;
					END_IF

				20:
					em.description 				:= 'Wait for close of own and neigbourflap';
					em.cmd.sc := TRUE;

			END_CASE

		ELSE
			em.cmd.sc := TRUE;

	END_CASE

END_ACTION
```

#### alarm.st
```iecst
ACTION alarm:

	// Open Time Too Long

	IF this.alarm.openTooLong.active AND NOT this.alarm.openTooLong.oldActive THEN
		this.alarm.openTooLong.instanceID := MpAlarmXSet(mpAlarmXCore, this.alarm.openTooLong.name);
	END_IF
	this.alarm.openTooLong.oldActive := this.alarm.openTooLong.active;

	// Close Time Too Long

	IF this.alarm.closeTooLong.active AND NOT this.alarm.closeTooLong.oldActive THEN
		this.alarm.closeTooLong.instanceID := MpAlarmXSet(mpAlarmXCore, this.alarm.closeTooLong.name);
	END_IF
	this.alarm.closeTooLong.oldActive := this.alarm.closeTooLong.active;

END_ACTION
```

#### upperFlap.st - Init, cyclic, exit code
```iecst
PROGRAM _INIT

	em.setup.name 			:= 'upperFlap';
	em.setup.parent.name 	:= 'wing';
	em.setup.reactTo 		:= BRDK_EM_REACT_TO_ALL;
	setupPointers;

	//Alarm texts
	this.alarm.closeTooLong.name := 'upperFlapCloseTooLong';
	this.alarm.openTooLong.name := 'upperFlapOpenTooLong';

END_PROGRAM

PROGRAM _CYCLIC

	setupPointers;
	ioMappingInput;

	// setup flap function block
	this.flap.enable 				:= TRUE;
	this.flap.cycleTime				:= em.status.cycleTime;
	this.flap.flapTime				:= interface.parameter.flapTime;
	this.flap.di_changeover 		:= this.hw.di_changeover;
	this.flap.simulation := gWingInterface.parameter.simulation;

	CASE em.mode OF
		MODE_PRODUCING,MODE_EMPTY: producing;
		MODE_MANUAL: testing;	// mode for testing flaps manually.
		ELSE em.cmd.sc := TRUE;
	END_CASE

	this.hw.do_open := this.flap.do_open;
	this.hmi.cycleTime := this.MTFilterMovingAverage_10.Out;

	IF gUpperFlapInterface.cmd.resetStatistics THEN
		gUpperFlapInterface.cmd.resetStatistics := FALSE;

		this.errBuffer_0.reset := TRUE;
		this.errBuffer_0();
		this.oldTeachingDone := FALSE;
		this.hmi.errorRate := 0;
		this.MTFilterMovingAverage_0(Enable:=FALSE);
		this.MTFilterMovingAverage_10(Enable:=FALSE);
		this.MTFilterMovingAverage_10_TMU(Enable:=FALSE);
	END_IF

	this.hmi.cycleTime := this.MTFilterMovingAverage_0.Out;				// moving avg of 40
	this.hmi.cycleTimeHMI := this.MTFilterMovingAverage_10.Out; 		// moving avg of 10
	this.hmi.cycleTimeTMU := this.MTFilterMovingAverage_10_TMU.Out;		// moving avg of 10

	alarm;

	em();
	this.flap();

	// FAT test
	CASE testStateFAT OF

		0:
			IF interface.cmd.wingTestManual THEN
				// Only execute if flap is closed
				IF this.hw.do_open=FALSE THEN
					interface.status.testResultFAT := FALSE; // reset result
					testStateFAT := 10;
				END_IF

			END_IF

		10:
			//wait 1s so flaps are closed before we start test.
			this.TON_test.IN := TRUE;
			this.TON_test.PT := T#500ms;
			this.TON_test();

			IF this.TON_test.Q THEN
				this.TON_test.IN := FALSE;
				this.TON_test();

				// Open flap
				this.flap.open := TRUE;
				testStateFAT := 20;
			END_IF

		20:
			IF this.flap.error THEN
				// Test fail
				testStateFAT := 60;
			ELSIF this.flap.position = FLAP_OPEN THEN
				testStateFAT 			:= 30;
			END_IF

		30:
			//wait 1s before closing
			this.TON_test.IN := TRUE;
			this.TON_test.PT := T#500ms;
			this.TON_test();

			IF this.TON_test.Q THEN
				this.TON_test.IN := FALSE;
				this.TON_test();

				// Close flap
				this.flap.close := TRUE;
				testStateFAT := 40;
			END_IF

		40:
			IF this.flap.error THEN
				// Test fail
				testStateFAT := 60;
			ELSIF this.flap.position = FLAP_CLOSED THEN
				testStateFAT 			:= 50;
			END_IF

		50:
			//wait 1s before closing
			this.TON_test.IN := TRUE;
			this.TON_test.PT := T#500ms;
			this.TON_test();

			IF this.TON_test.Q THEN
				this.TON_test.IN := FALSE;
				this.TON_test();

				interface.status.testResultFAT := TRUE; // Good result
				testStateFAT := 60;
			END_IF

		60:
			// Reset error (if any) before finishing test
			this.flap.resetError := this.flap.error;

			IF NOT this.flap.error THEN
				interface.cmd.wingTestManual := FALSE; // signal test done

				// Start next test (we are done here)
				gMiddleFlapInterface.cmd.wingTestManual := TRUE;
				testStateFAT := 0;
			END_IF

	END_CASE

END_PROGRAM

PROGRAM _EXIT
	this.MTFilterMovingAverage_0(Enable:=FALSE);
	this.MTFilterMovingAverage_10(Enable:=FALSE);
	this.MTFilterMovingAverage_10_TMU(Enable:=FALSE);
END_PROGRAM
```

#### ioMappingInput.st
```iecst
ACTION ioMappingInput:

	IF this.hwWu[0].di_wingUnitActive THEN
		this.flap.WUstepperConnected := TRUE;
		this.flap.positionFromWUstepper := this.hwWu[0].flapPosition;
	ELSIF this.hwWu[1].di_wingUnitActive THEN
		this.flap.WUstepperConnected := TRUE;
		this.flap.positionFromWUstepper := this.hwWu[1].flapPosition;
	ELSE
		this.flap.WUstepperConnected := FALSE;
	END_IF

	gWingInterface.status.stepperWUConnected	:= this.hwWu[0].di_wingUnitActive OR this.hwWu[1].di_wingUnitActive;

END_ACTION
```

#### testing.st
```iecst
ACTION testing:

	this.flapTest.openTime := this.flap.openTimeAfterChangeover;
	this.flapTest.closingTime := this.flap.closingTimeAfterChangeover;
	this.flapTest.openTimeOK := this.flapTest.openTime >= 210 AND this.flapTest.openTime <= 230;
	this.flapTest.closingTimeOK := this.flapTest.closingTime >= 210 AND this.flapTest.closingTime <= 230;

	CASE this.test.state OF

		0:
			IF NOT interface.cmd.manuelMode THEN
				interface.cmd.runFlapContinuously := FALSE;
				em.substate := 0; // go back to 0 (no more manuel mode)
			ELSIF gWingInterface.status.startTestSequence THEN
				interface.cmd.runFlapContinuously := FALSE; // can't run while doing test sequence.
				this.test.state := 10;
			ELSIF interface.cmd.runFlapContinuously THEN
				this.test.state := 60;
			END_IF

			(**** Run sequence ****)

		10:
			IF NOT gWingInterface.status.startTestSequence THEN
				this.test.state := 0;
			ELSIF interface.cmd.open THEN
				this.flap.open := TRUE;
				this.test.state := 20;
			END_IF

		20:

			IF this.flap.error THEN
				this.alarm.openTooLong.active := TRUE;
			ELSIF this.flap.position = FLAP_OPEN THEN
				this.time.elapsed := 0;
				this.test.state := 30;
			END_IF

		30:
			this.time.elapsed := this.time.elapsed + em.status.cycleTime;
			IF this.time.elapsed >= this.flapTest.waitTime THEN
				this.flap.close := TRUE;		// close cmd
				this.test.state := 40;
			END_IF

		40:
			IF this.flap.error THEN
				this.alarm.closeTooLong.active := TRUE;
			ELSIF this.flap.position = FLAP_CLOSED THEN
				this.time.elapsed := 0;
				this.test.state := 50;
			END_IF

		50:
			em.description := 'Wait delay before opening next flap';

			this.time.elapsed := this.time.elapsed + em.status.cycleTime;
			IF this.time.elapsed >= this.flapTest.waitTime THEN
				interface.cmd.open := FALSE;	// Will signal to wing that flap is done with open/close.
				this.test.state := 10;
			END_IF

			(**** Run continously ****)

		60:
			IF NOT interface.cmd.runFlapContinuously THEN
				this.test.state := 0;
			ELSE
				this.flap.open := TRUE;
				this.test.state := 70;
			END_IF

		70:
			IF this.flap.error THEN
				this.alarm.openTooLong.active := TRUE;
			ELSIF this.flap.position = FLAP_OPEN THEN
				this.time.elapsed := 0;
				this.test.state := 80;
			END_IF

		80:
			this.time.elapsed := this.time.elapsed + em.status.cycleTime;
			IF this.time.elapsed >= this.flapTest.waitTime THEN
				this.flap.close := TRUE;		// close cmd
				this.test.state := 90;
			END_IF

		90:
			IF this.flap.error THEN
				this.alarm.closeTooLong.active := TRUE;
			ELSIF this.flap.position = FLAP_CLOSED THEN
				this.time.elapsed := 0;
				this.test.state := 100;
			END_IF

		100:
			this.time.elapsed := this.time.elapsed + em.status.cycleTime;
			IF this.time.elapsed >= this.flapTest.waitTime THEN
				this.test.state := 60;
			END_IF

	END_CASE

END_ACTION
```

#### setupPointers.st
```iecst
ACTION setupPointers:
	interface ACCESS ADR(gUpperFlapInterface);
END_ACTION
```

#### local.typ - Local data types
```iecst
TYPE
	local_typ : 	STRUCT
		time : local_time_typ;
		waitingTime : waiting_time_typ;
		flap : legoCM20Flap;
		alarm : local_alarm_typ;
		hwAir : local_hw_typ;
		hw : local_hw_typ;
		hwWu : ARRAY[0..1]OF wu20_typ; (*Communication with wing unit*)
		flapTest : flapTest_typ;
		hmi : local_hmi_typ;
		afterCount : BOOL;
		rejectNext : BOOL;
		cycleTimeTheoretical : UDINT;
		test : local_test_typ;
		errBuffer_0 : errBuffer;
		previousState : UINT;
		oldTeachingDone : BOOL;
		upperFlapCycleTime : UDINT;
		MTFilterMovingAverage_0 : MTFilterMovingAverage;
		MTFilterMovingAverage_10 : MTFilterMovingAverage;
		MTFilterMovingAverage_10_TMU : MTFilterMovingAverage;
		lastUpperFlapCycleTime : UDINT;
		TON_test : TON;
	END_STRUCT;
	local_hmi_typ : 	STRUCT
		errorRate : REAL;
		cycleTime : REAL; (*moving avg of 40*)
		cycleTimeHMI : REAL; (*moving avg of 10*)
		cycleTimeTMU : REAL;
		cycleTimeRaw : REAL;
		rejectAll : BOOL;
	END_STRUCT;
	wu20_typ : 	STRUCT
		flapPosition : DINT; (*4 = open, 8 = closed*)
		di_wingUnitActive : BOOL;
	END_STRUCT;
	waiting_time_typ : 	STRUCT
		current : UDINT; (*[us]*)
		average : UDINT; (*[us]*)
		count : USINT;
	END_STRUCT;
	local_hw_typ : 	STRUCT
		di_changeover : BOOL;
		do_open : BOOL;
	END_STRUCT;
	local_alarm_typ : 	STRUCT
		openTooLong : gAlarm_struct_typ;
		closeTooLong : gAlarm_struct_typ;
	END_STRUCT;
	flapTest_typ : 	STRUCT
		flapSequenceTest : BOOL; (*Flaps will run in a sequence (usually over night)*)
		openTime : UDINT;
		closingTime : UDINT;
		waitTime : UDINT := 200000;
		alarmOpenTooLong : BOOL;
		alarmCloseTooLong : BOOL;
		openTimeOK : BOOL;
		closingTimeOK : BOOL;
	END_STRUCT;
	local_test_typ : 	STRUCT
		state : USINT;
	END_STRUCT;
END_TYPE
```

#### local.var - Local variables
```iecst
VAR
	interface : REFERENCE TO gUpperFlapInterface_typ;
	this : {REDUND_UNREPLICABLE} local_typ;
	em : {REDUND_UNREPLICABLE} brdkEM;
END_VAR
VAR CONSTANT
	ERR_BUFFER_SIZE : UINT := 99;
END_VAR
VAR
	testAfterCount : BOOL;
	testStateFAT : USINT;
END_VAR
```

#### LocalFunctions.fun
```iecst
FUNCTION_BLOCK errBuffer (*LIFO buffer to save the status of last 100 portions and calculate the error rate*)
	VAR_INPUT
		input : BOOL; (*input (OK or not OK)*)
		array : {REDUND_UNREPLICABLE} ARRAY[0..ERR_BUFFER_SIZE] OF BOOL := [100(TRUE)];
		pushToBuffer : BOOL; (*push input to buffer*)
		reset : BOOL := FALSE;
	END_VAR
	VAR_OUTPUT
		errorRate : REAL;
	END_VAR
	VAR
		idx : UINT;
		okItems : REAL;
		itemsInBuffer : UINT;
	END_VAR
END_FUNCTION_BLOCK
```

#### errBuffer.st
```iecst
(* TODO: Add your comment here *)
FUNCTION_BLOCK errBuffer
	IF pushToBuffer THEN

		// Move full array 1 idx down (stack push implementation).
		memmove(ADR(array[1]), ADR(array[0]), SIZEOF(array[0])*ERR_BUFFER_SIZE);
		array[0] := input;

		// Limit items by the size of the buffer
		itemsInBuffer := itemsInBuffer + 1;
		IF itemsInBuffer > ERR_BUFFER_SIZE+1 THEN
			itemsInBuffer := ERR_BUFFER_SIZE+1;
		END_IF

		// Calculate error rate
		okItems := 0;
		FOR idx := 0 TO (itemsInBuffer-1) DO
			IF array[idx] = TRUE THEN
				okItems := okItems + 1;
			END_IF;
		END_FOR;
		errorRate := 1.0 - (okItems / UINT_TO_REAL(itemsInBuffer));
		pushToBuffer := FALSE;

	END_IF

	IF reset THEN
		reset := FALSE;

		errorRate := 0;
		memset(ADR(array),1,SIZEOF(array));
		idx := 0;
		okItems := 0;
		itemsInBuffer := ERR_BUFFER_SIZE+1;

	END_IF

END_FUNCTION_BLOCK
```

### upperFlapGlobal.typ
```iecst
TYPE
	gUpperFlapInterface_status_typ : 	STRUCT
		ready : BOOL;
		request : BOOL;
		openCloseTime : UDINT;
		active : BOOL;
		countAftercount : UDINT;
		OKPortions : UDINT;
		NOKPortions : UDINT;
		lastCycleTime : UDINT;
		testResultFAT : BOOL; (*TRUE=good, FALSE=bad*)
	END_STRUCT;
	gUpperFlapInterface_para_typ : 	STRUCT
		brickStatus : gFlap_brick_status_typ;
		openTime : UDINT; (*Time the flap stays open*)
		flapTime : UDINT; (*Time that the flap is to open or close*)
		startBeltWaitTime : UDINT;
	END_STRUCT;
	gUpperFlapInterface_cmd_typ : 	STRUCT
		start : BOOL;
		runFlapContinuously : BOOL;
		open : BOOL; (*wing -> flap to open doing sequence test*)
		brickStatusReady : BOOL;
		manuelMode : BOOL;
		resetStatistics : BOOL;
		wingTestManual : BOOL;
	END_STRUCT;
	gUpperFlapInterface_typ : 	STRUCT
		cmd : gUpperFlapInterface_cmd_typ;
		parameter : gUpperFlapInterface_para_typ;
		status : gUpperFlapInterface_status_typ;
	END_STRUCT;
END_TYPE
```

### upperFlapGlobal.var
```iecst
VAR
	gUpperFlapInterface : gUpperFlapInterface_typ;
END_VAR
```

### Program Logical/modules/main/wing/middleFlap/middleFlap (IEC)
